// TIA Portal project "BangTai" (V17)

(* hardware
DEVICE "S7-1200 station_1"  S7-1200 Station
   slot 0: "Rack_0"  S7-1200 Rack  Rack  V1.0
   slot 1: "PLC _1"  CPU 1214C AC/DC/Rly  6ES7 214-1BG40-0XB0  V4.5
*)

// ===== PLC "PLC _1"  CPU 1214C AC/DC/Rly =====

VAR_GLOBAL   // PLC tag table "AO"
   "AQ_WeighConveyor.SpeedCMD" AT %QW0 : Int;
   "AQ_NormalConveyor.SpeedCMD" AT %QW2 : Int;
END_VAR

VAR_GLOBAL   // PLC tag table "AI"
   "AI_Weigh" AT %IW0 : Int;
   "AI_WeighConveyor.Speed" AT %IW2 : Int;
   "AI_NormalConveyor" AT %IW4 : Int;
END_VAR

VAR_GLOBAL   // PLC tag table "DO"
   "DO_WeighConveyor.CMD" AT %I7.0 : Bool;
   "DO_NormalConveyor.CMD" AT %I7.1 : Bool;
END_VAR

VAR_GLOBAL   // PLC tag table "DI"
   "DI_WeighConveyor.Run" AT %I6.0 : Bool;
   "DI_WeighConveyor.Fault" AT %I6.1 : Bool;
   "DI_WeighConveyor.Remote" AT %I6.2 : Bool;
   "DI_NormalConveyor.Run" AT %I6.3 : Bool;
   "DI_NormalConveyor.Fault" AT %I6.4 : Bool;
   "DI_NormalConveyor.Remote" AT %I6.5 : Bool;
   "DI_Oject" AT %I6.6 : Bool;
   "DI_WrongObject" AT %I6.7 : Bool;
END_VAR

TYPE "Sensor"
   STRUCT
      High_Value : Real;
      Low_Value : Real;
      Ratio : Real;
      Bias : Real;
      Real_Value : Real;
      HLM : Real;
      LLM : Real;
      HLM_Auxiliary : Real;
      LLM_Auxiliary : Real;
      Input_Error : Bool;
      Sensor_Error : Bool;
      Alarm_HLM : Bool;
      Alarm_LLM : Bool;
   END_STRUCT;
END_TYPE

TYPE "Motor_VDF"
   STRUCT
      Ctrl_Mode : Int;   // 0-Stop; 1-Manual; 2-Auto
      Enable : Bool;
      Lock : Bool;
      Manual_Lock : Bool;
      Status : Int;
      Runtime_60s : Int;
      Runtime_h : Int;
      Runtime_m : Int;
      Runtime_s : Int;
      P : Real;
      I : Real;
      D : Real;
      "Speed.RealValue" : Real;   // Gia tri doc tu bien tan
      "Speed.WriteHLM(Hz)" : Real;   // Gia tri tan so out Low
      "Speed.WriteLLM(Hz)" : Real;   // Gia tri tan so out High
      "Speed.Manual(Hz)" : Real;   // Gia tri tan so chay tay
      "Speed.WriteHLM(%)" : Real;   // Gia tri dung cho khoi PID 0->100 %
      "Speed.WriteLLM(%)" : Real;   // Gia tri tan so out High
      "Speed.Manual(%)" : Real;   // Gia tri tan so chay tay
      "ReadSpeed.Ratio" : Real;
      "ReadSpeed.Bias" : Real;
   END_STRUCT;
END_TYPE

TYPE "Motor_Normal"
   STRUCT
      Ctrl_Mode : Int;   // 0-Stop; 1-Manual; 2-Auto
      Enable : Bool;
      Lock : Bool;
      Manual_Lock : Bool;
      Status : Int;   // -1: Fault, 0:Stop, 1:Run
      Runtime_60s : Int;
      Runtime_h : Int;
      Runtime_m : Int;
      Runtime_s : Int;
   END_STRUCT;
END_TYPE

// folder: DataBlock

DATA_BLOCK "DB_READ_ABALOG"   // DB1
{ S7_Optimized_Access := 'TRUE' }
VERSION : 0.1
   VAR
      Weigh : "Sensor";
      sensor_weigh : Bool;
      sensor_wrong_object : Bool;
   END_VAR
BEGIN
END_DATA_BLOCK

DATA_BLOCK "DB_Conveyor"   // DB2
{ S7_Optimized_Access := 'TRUE' }
VERSION : 0.1
   VAR
      weigh_conveyor : "Motor_VDF";
      normal_conveyor : "Motor_VDF";
   END_VAR
BEGIN
END_DATA_BLOCK

// folder: (top level)

FUNCTION "FC_READ_ANALOG" : Void   // FC2, LAD
{ S7_Optimized_Access := 'TRUE' }
VERSION : 0.1
BEGIN

REGION Network 1: Đọc giá trị tốc độ băng tải cân
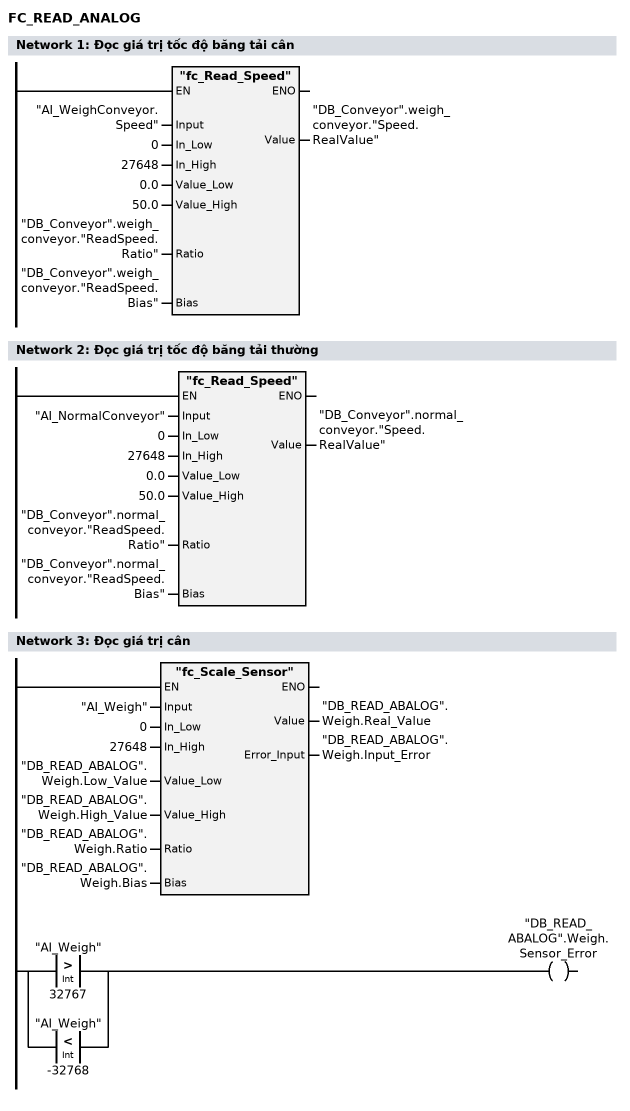
   RUNG wire#powerrail
      "fc_Read_Speed"(Input := "AI_WeighConveyor.Speed", In_Low := 0, In_High := 27648, Value_Low := 0.0, Value_High := 50.0, Ratio := "DB_Conveyor".weigh_conveyor."ReadSpeed.Ratio", Bias := "DB_Conveyor".weigh_conveyor."ReadSpeed.Bias", Value => "DB_Conveyor".weigh_conveyor."Speed.RealValue")
   END_RUNG
   // the same network as SCL:
   "fc_Read_Speed"(Input := "AI_WeighConveyor.Speed",
                   In_Low := 0,
                   In_High := 27648,
                   Value_Low := 0.0,
                   Value_High := 50.0,
                   Ratio := "DB_Conveyor".weigh_conveyor."ReadSpeed.Ratio",
                   Bias := "DB_Conveyor".weigh_conveyor."ReadSpeed.Bias",
                   Value => "DB_Conveyor".weigh_conveyor."Speed.RealValue");
END_REGION

REGION Network 2: Đọc giá trị tốc độ băng tải thường
   RUNG wire#powerrail
      "fc_Read_Speed"(Input := "AI_NormalConveyor", In_Low := 0, In_High := 27648, Value_Low := 0.0, Value_High := 50.0, Ratio := "DB_Conveyor".normal_conveyor."ReadSpeed.Ratio", Bias := "DB_Conveyor".normal_conveyor."ReadSpeed.Bias", Value => "DB_Conveyor".normal_conveyor."Speed.RealValue")
   END_RUNG
   // the same network as SCL:
   "fc_Read_Speed"(Input := "AI_NormalConveyor",
                   In_Low := 0,
                   In_High := 27648,
                   Value_Low := 0.0,
                   Value_High := 50.0,
                   Ratio := "DB_Conveyor".normal_conveyor."ReadSpeed.Ratio",
                   Bias := "DB_Conveyor".normal_conveyor."ReadSpeed.Bias",
                   Value => "DB_Conveyor".normal_conveyor."Speed.RealValue");
END_REGION

REGION Network 3: Đọc giá trị cân
   RUNG wire#powerrail
      "fc_Scale_Sensor"(Input := "AI_Weigh", In_Low := 0, In_High := 27648, Value_Low := "DB_READ_ABALOG".Weigh.Low_Value, Value_High := "DB_READ_ABALOG".Weigh.High_Value, Ratio := "DB_READ_ABALOG".Weigh.Ratio, Bias := "DB_READ_ABALOG".Weigh.Bias, Value => "DB_READ_ABALOG".Weigh.Real_Value, Error_Input => "DB_READ_ABALOG".Weigh.Input_Error)
   END_RUNG
   RUNG wire#powerrail
      { S7_Templates := "SrcType := Int" } GT_Contact(in1 := "AI_Weigh", in2 := 32767)
      wire#w1
      Coil( "DB_READ_ABALOG".Weigh.Sensor_Error )
   END_RUNG
   RUNG wire#powerrail
      { S7_Templates := "SrcType := Int" } LT_Contact(in1 := "AI_Weigh", in2 := -32768)
   END_RUNG wire#w1
   // the same network as SCL:
   "fc_Scale_Sensor"(Input := "AI_Weigh",
                     In_Low := 0,
                     In_High := 27648,
                     Value_Low := "DB_READ_ABALOG".Weigh.Low_Value,
                     Value_High := "DB_READ_ABALOG".Weigh.High_Value,
                     Ratio := "DB_READ_ABALOG".Weigh.Ratio,
                     Bias := "DB_READ_ABALOG".Weigh.Bias,
                     Value => "DB_READ_ABALOG".Weigh.Real_Value,
                     Error_Input => "DB_READ_ABALOG".Weigh.Input_Error);
   "DB_READ_ABALOG".Weigh.Sensor_Error := ("AI_Weigh" > 32767) OR ("AI_Weigh" < (-32768));
END_REGION
END_FUNCTION

FUNCTION "FC_ALARM" : Void   // FC3, LAD
{ S7_Optimized_Access := 'TRUE' }
VERSION : 0.1
BEGIN

REGION Network 1: Canh bao ap suat buong dot cao
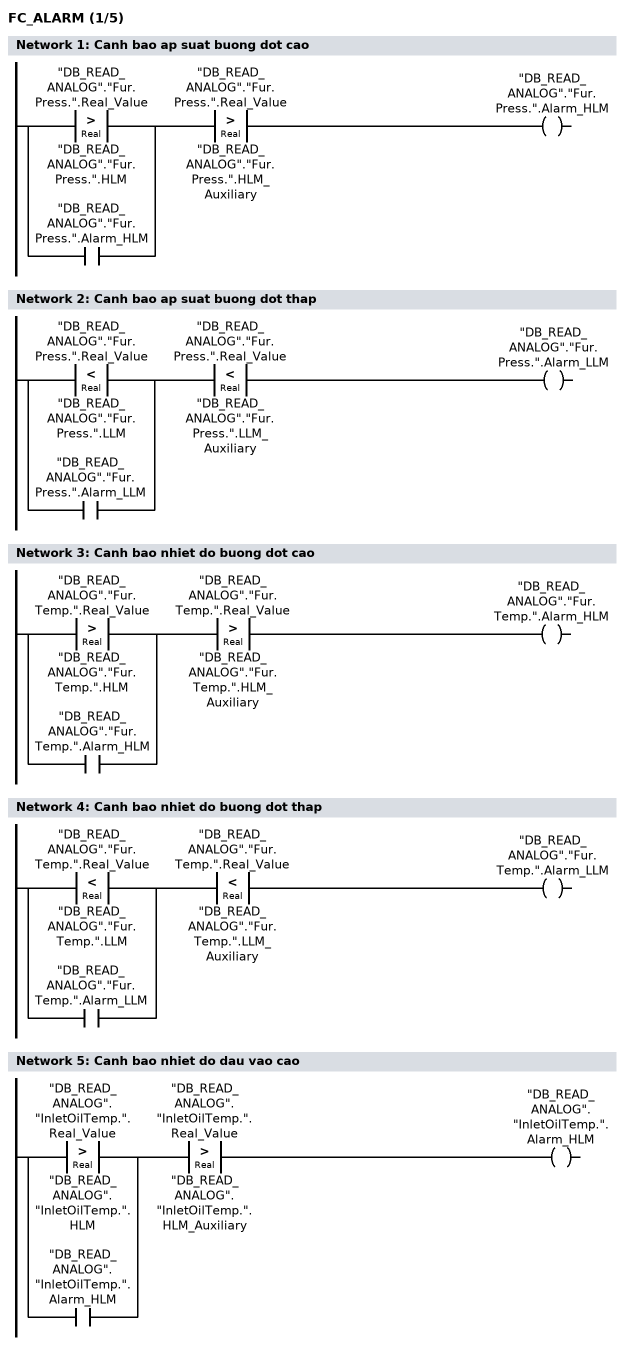
   RUNG wire#powerrail
      { S7_Templates := "SrcType := Real" } GT_Contact(in1 := "DB_READ_ANALOG"."Fur.Press.".Real_Value, in2 := "DB_READ_ANALOG"."Fur.Press.".HLM)
      wire#w1
      { S7_Templates := "SrcType := Real" } GT_Contact(in1 := "DB_READ_ANALOG"."Fur.Press.".Real_Value, in2 := "DB_READ_ANALOG"."Fur.Press.".HLM_Auxiliary)
      Coil( "DB_READ_ANALOG"."Fur.Press.".Alarm_HLM )
   END_RUNG
   RUNG wire#powerrail
      Contact( "DB_READ_ANALOG"."Fur.Press.".Alarm_HLM )
   END_RUNG wire#w1
   // the same network as SCL:
   "DB_READ_ANALOG"."Fur.Press.".Alarm_HLM := (("DB_READ_ANALOG"."Fur.Press.".Real_Value > "DB_READ_ANALOG"."Fur.Press.".HLM) OR "DB_READ_ANALOG"."Fur.Press.".Alarm_HLM) AND ("DB_READ_ANALOG"."Fur.Press.".Real_Value > "DB_READ_ANALOG"."Fur.Press.".HLM_Auxiliary);
END_REGION

REGION Network 2: Canh bao ap suat buong dot thap
   RUNG wire#powerrail
      { S7_Templates := "SrcType := Real" } LT_Contact(in1 := "DB_READ_ANALOG"."Fur.Press.".Real_Value, in2 := "DB_READ_ANALOG"."Fur.Press.".LLM)
      wire#w1
      { S7_Templates := "SrcType := Real" } LT_Contact(in1 := "DB_READ_ANALOG"."Fur.Press.".Real_Value, in2 := "DB_READ_ANALOG"."Fur.Press.".LLM_Auxiliary)
      Coil( "DB_READ_ANALOG"."Fur.Press.".Alarm_LLM )
   END_RUNG
   RUNG wire#powerrail
      Contact( "DB_READ_ANALOG"."Fur.Press.".Alarm_LLM )
   END_RUNG wire#w1
   // the same network as SCL:
   "DB_READ_ANALOG"."Fur.Press.".Alarm_LLM := (("DB_READ_ANALOG"."Fur.Press.".Real_Value < "DB_READ_ANALOG"."Fur.Press.".LLM) OR "DB_READ_ANALOG"."Fur.Press.".Alarm_LLM) AND ("DB_READ_ANALOG"."Fur.Press.".Real_Value < "DB_READ_ANALOG"."Fur.Press.".LLM_Auxiliary);
END_REGION

REGION Network 3: Canh bao nhiet do buong dot cao
   RUNG wire#powerrail
      { S7_Templates := "SrcType := Real" } GT_Contact(in1 := "DB_READ_ANALOG"."Fur.Temp.".Real_Value, in2 := "DB_READ_ANALOG"."Fur.Temp.".HLM)
      wire#w1
      { S7_Templates := "SrcType := Real" } GT_Contact(in1 := "DB_READ_ANALOG"."Fur.Temp.".Real_Value, in2 := "DB_READ_ANALOG"."Fur.Temp.".HLM_Auxiliary)
      Coil( "DB_READ_ANALOG"."Fur.Temp.".Alarm_HLM )
   END_RUNG
   RUNG wire#powerrail
      Contact( "DB_READ_ANALOG"."Fur.Temp.".Alarm_HLM )
   END_RUNG wire#w1
   // the same network as SCL:
   "DB_READ_ANALOG"."Fur.Temp.".Alarm_HLM := (("DB_READ_ANALOG"."Fur.Temp.".Real_Value > "DB_READ_ANALOG"."Fur.Temp.".HLM) OR "DB_READ_ANALOG"."Fur.Temp.".Alarm_HLM) AND ("DB_READ_ANALOG"."Fur.Temp.".Real_Value > "DB_READ_ANALOG"."Fur.Temp.".HLM_Auxiliary);
END_REGION

REGION Network 4: Canh bao nhiet do buong dot thap
   RUNG wire#powerrail
      { S7_Templates := "SrcType := Real" } LT_Contact(in1 := "DB_READ_ANALOG"."Fur.Temp.".Real_Value, in2 := "DB_READ_ANALOG"."Fur.Temp.".LLM)
      wire#w1
      { S7_Templates := "SrcType := Real" } LT_Contact(in1 := "DB_READ_ANALOG"."Fur.Temp.".Real_Value, in2 := "DB_READ_ANALOG"."Fur.Temp.".LLM_Auxiliary)
      Coil( "DB_READ_ANALOG"."Fur.Temp.".Alarm_LLM )
   END_RUNG
   RUNG wire#powerrail
      Contact( "DB_READ_ANALOG"."Fur.Temp.".Alarm_LLM )
   END_RUNG wire#w1
   // the same network as SCL:
   "DB_READ_ANALOG"."Fur.Temp.".Alarm_LLM := (("DB_READ_ANALOG"."Fur.Temp.".Real_Value < "DB_READ_ANALOG"."Fur.Temp.".LLM) OR "DB_READ_ANALOG"."Fur.Temp.".Alarm_LLM) AND ("DB_READ_ANALOG"."Fur.Temp.".Real_Value < "DB_READ_ANALOG"."Fur.Temp.".LLM_Auxiliary);
END_REGION

REGION Network 5: Canh bao nhiet do dau vao cao
   RUNG wire#powerrail
      { S7_Templates := "SrcType := Real" } GT_Contact(in1 := "DB_READ_ANALOG"."InletOilTemp.".Real_Value, in2 := "DB_READ_ANALOG"."InletOilTemp.".HLM)
      wire#w1
      { S7_Templates := "SrcType := Real" } GT_Contact(in1 := "DB_READ_ANALOG"."InletOilTemp.".Real_Value, in2 := "DB_READ_ANALOG"."InletOilTemp.".HLM_Auxiliary)
      Coil( "DB_READ_ANALOG"."InletOilTemp.".Alarm_HLM )
   END_RUNG
   RUNG wire#powerrail
      Contact( "DB_READ_ANALOG"."InletOilTemp.".Alarm_HLM )
   END_RUNG wire#w1
   // the same network as SCL:
   "DB_READ_ANALOG"."InletOilTemp.".Alarm_HLM := (("DB_READ_ANALOG"."InletOilTemp.".Real_Value > "DB_READ_ANALOG"."InletOilTemp.".HLM) OR "DB_READ_ANALOG"."InletOilTemp.".Alarm_HLM) AND ("DB_READ_ANALOG"."InletOilTemp.".Real_Value > "DB_READ_ANALOG"."InletOilTemp.".HLM_Auxiliary);
END_REGION

REGION Network 6: Canh bao nhiet do dau vao thap
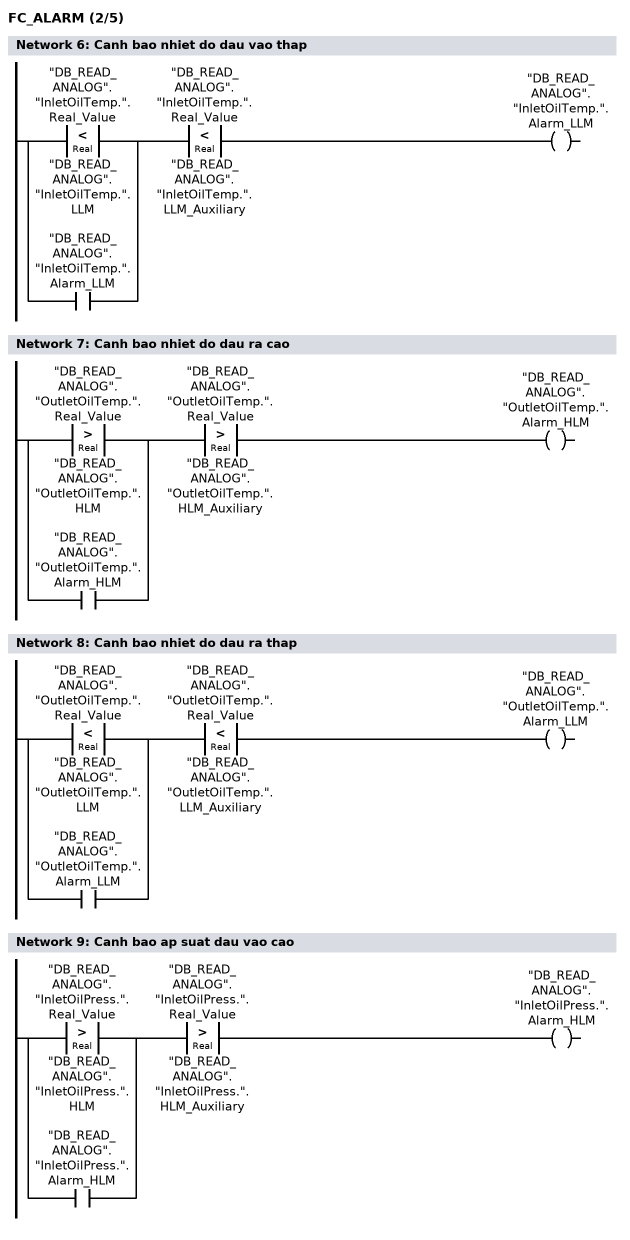
   RUNG wire#powerrail
      { S7_Templates := "SrcType := Real" } LT_Contact(in1 := "DB_READ_ANALOG"."InletOilTemp.".Real_Value, in2 := "DB_READ_ANALOG"."InletOilTemp.".LLM)
      wire#w1
      { S7_Templates := "SrcType := Real" } LT_Contact(in1 := "DB_READ_ANALOG"."InletOilTemp.".Real_Value, in2 := "DB_READ_ANALOG"."InletOilTemp.".LLM_Auxiliary)
      Coil( "DB_READ_ANALOG"."InletOilTemp.".Alarm_LLM )
   END_RUNG
   RUNG wire#powerrail
      Contact( "DB_READ_ANALOG"."InletOilTemp.".Alarm_LLM )
   END_RUNG wire#w1
   // the same network as SCL:
   "DB_READ_ANALOG"."InletOilTemp.".Alarm_LLM := (("DB_READ_ANALOG"."InletOilTemp.".Real_Value < "DB_READ_ANALOG"."InletOilTemp.".LLM) OR "DB_READ_ANALOG"."InletOilTemp.".Alarm_LLM) AND ("DB_READ_ANALOG"."InletOilTemp.".Real_Value < "DB_READ_ANALOG"."InletOilTemp.".LLM_Auxiliary);
END_REGION

REGION Network 7: Canh bao nhiet do dau ra cao
   RUNG wire#powerrail
      { S7_Templates := "SrcType := Real" } GT_Contact(in1 := "DB_READ_ANALOG"."OutletOilTemp.".Real_Value, in2 := "DB_READ_ANALOG"."OutletOilTemp.".HLM)
      wire#w1
      { S7_Templates := "SrcType := Real" } GT_Contact(in1 := "DB_READ_ANALOG"."OutletOilTemp.".Real_Value, in2 := "DB_READ_ANALOG"."OutletOilTemp.".HLM_Auxiliary)
      Coil( "DB_READ_ANALOG"."OutletOilTemp.".Alarm_HLM )
   END_RUNG
   RUNG wire#powerrail
      Contact( "DB_READ_ANALOG"."OutletOilTemp.".Alarm_HLM )
   END_RUNG wire#w1
   // the same network as SCL:
   "DB_READ_ANALOG"."OutletOilTemp.".Alarm_HLM := (("DB_READ_ANALOG"."OutletOilTemp.".Real_Value > "DB_READ_ANALOG"."OutletOilTemp.".HLM) OR "DB_READ_ANALOG"."OutletOilTemp.".Alarm_HLM) AND ("DB_READ_ANALOG"."OutletOilTemp.".Real_Value > "DB_READ_ANALOG"."OutletOilTemp.".HLM_Auxiliary);
END_REGION

REGION Network 8: Canh bao nhiet do dau ra thap
   RUNG wire#powerrail
      { S7_Templates := "SrcType := Real" } LT_Contact(in1 := "DB_READ_ANALOG"."OutletOilTemp.".Real_Value, in2 := "DB_READ_ANALOG"."OutletOilTemp.".LLM)
      wire#w1
      { S7_Templates := "SrcType := Real" } LT_Contact(in1 := "DB_READ_ANALOG"."OutletOilTemp.".Real_Value, in2 := "DB_READ_ANALOG"."OutletOilTemp.".LLM_Auxiliary)
      Coil( "DB_READ_ANALOG"."OutletOilTemp.".Alarm_LLM )
   END_RUNG
   RUNG wire#powerrail
      Contact( "DB_READ_ANALOG"."OutletOilTemp.".Alarm_LLM )
   END_RUNG wire#w1
   // the same network as SCL:
   "DB_READ_ANALOG"."OutletOilTemp.".Alarm_LLM := (("DB_READ_ANALOG"."OutletOilTemp.".Real_Value < "DB_READ_ANALOG"."OutletOilTemp.".LLM) OR "DB_READ_ANALOG"."OutletOilTemp.".Alarm_LLM) AND ("DB_READ_ANALOG"."OutletOilTemp.".Real_Value < "DB_READ_ANALOG"."OutletOilTemp.".LLM_Auxiliary);
END_REGION

REGION Network 9: Canh bao ap suat dau vao cao
   RUNG wire#powerrail
      { S7_Templates := "SrcType := Real" } GT_Contact(in1 := "DB_READ_ANALOG"."InletOilPress.".Real_Value, in2 := "DB_READ_ANALOG"."InletOilPress.".HLM)
      wire#w1
      { S7_Templates := "SrcType := Real" } GT_Contact(in1 := "DB_READ_ANALOG"."InletOilPress.".Real_Value, in2 := "DB_READ_ANALOG"."InletOilPress.".HLM_Auxiliary)
      Coil( "DB_READ_ANALOG"."InletOilPress.".Alarm_HLM )
   END_RUNG
   RUNG wire#powerrail
      Contact( "DB_READ_ANALOG"."InletOilPress.".Alarm_HLM )
   END_RUNG wire#w1
   // the same network as SCL:
   "DB_READ_ANALOG"."InletOilPress.".Alarm_HLM := (("DB_READ_ANALOG"."InletOilPress.".Real_Value > "DB_READ_ANALOG"."InletOilPress.".HLM) OR "DB_READ_ANALOG"."InletOilPress.".Alarm_HLM) AND ("DB_READ_ANALOG"."InletOilPress.".Real_Value > "DB_READ_ANALOG"."InletOilPress.".HLM_Auxiliary);
END_REGION

REGION Network 10: Canh bao ap suat dau vao thap
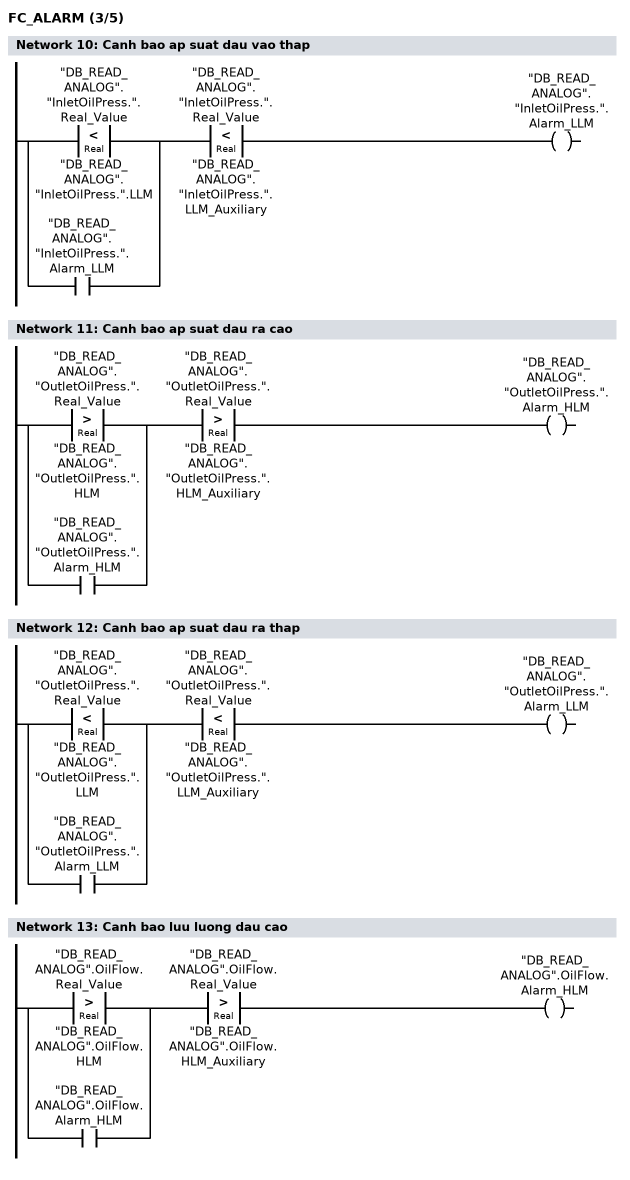
   RUNG wire#powerrail
      { S7_Templates := "SrcType := Real" } LT_Contact(in1 := "DB_READ_ANALOG"."InletOilPress.".Real_Value, in2 := "DB_READ_ANALOG"."InletOilPress.".LLM)
      wire#w1
      { S7_Templates := "SrcType := Real" } LT_Contact(in1 := "DB_READ_ANALOG"."InletOilPress.".Real_Value, in2 := "DB_READ_ANALOG"."InletOilPress.".LLM_Auxiliary)
      Coil( "DB_READ_ANALOG"."InletOilPress.".Alarm_LLM )
   END_RUNG
   RUNG wire#powerrail
      Contact( "DB_READ_ANALOG"."InletOilPress.".Alarm_LLM )
   END_RUNG wire#w1
   // the same network as SCL:
   "DB_READ_ANALOG"."InletOilPress.".Alarm_LLM := (("DB_READ_ANALOG"."InletOilPress.".Real_Value < "DB_READ_ANALOG"."InletOilPress.".LLM) OR "DB_READ_ANALOG"."InletOilPress.".Alarm_LLM) AND ("DB_READ_ANALOG"."InletOilPress.".Real_Value < "DB_READ_ANALOG"."InletOilPress.".LLM_Auxiliary);
END_REGION

REGION Network 11: Canh bao ap suat dau ra cao
   RUNG wire#powerrail
      { S7_Templates := "SrcType := Real" } GT_Contact(in1 := "DB_READ_ANALOG"."OutletOilPress.".Real_Value, in2 := "DB_READ_ANALOG"."OutletOilPress.".HLM)
      wire#w1
      { S7_Templates := "SrcType := Real" } GT_Contact(in1 := "DB_READ_ANALOG"."OutletOilPress.".Real_Value, in2 := "DB_READ_ANALOG"."OutletOilPress.".HLM_Auxiliary)
      Coil( "DB_READ_ANALOG"."OutletOilPress.".Alarm_HLM )
   END_RUNG
   RUNG wire#powerrail
      Contact( "DB_READ_ANALOG"."OutletOilPress.".Alarm_HLM )
   END_RUNG wire#w1
   // the same network as SCL:
   "DB_READ_ANALOG"."OutletOilPress.".Alarm_HLM := (("DB_READ_ANALOG"."OutletOilPress.".Real_Value > "DB_READ_ANALOG"."OutletOilPress.".HLM) OR "DB_READ_ANALOG"."OutletOilPress.".Alarm_HLM) AND ("DB_READ_ANALOG"."OutletOilPress.".Real_Value > "DB_READ_ANALOG"."OutletOilPress.".HLM_Auxiliary);
END_REGION

REGION Network 12: Canh bao ap suat dau ra thap
   RUNG wire#powerrail
      { S7_Templates := "SrcType := Real" } LT_Contact(in1 := "DB_READ_ANALOG"."OutletOilPress.".Real_Value, in2 := "DB_READ_ANALOG"."OutletOilPress.".LLM)
      wire#w1
      { S7_Templates := "SrcType := Real" } LT_Contact(in1 := "DB_READ_ANALOG"."OutletOilPress.".Real_Value, in2 := "DB_READ_ANALOG"."OutletOilPress.".LLM_Auxiliary)
      Coil( "DB_READ_ANALOG"."OutletOilPress.".Alarm_LLM )
   END_RUNG
   RUNG wire#powerrail
      Contact( "DB_READ_ANALOG"."OutletOilPress.".Alarm_LLM )
   END_RUNG wire#w1
   // the same network as SCL:
   "DB_READ_ANALOG"."OutletOilPress.".Alarm_LLM := (("DB_READ_ANALOG"."OutletOilPress.".Real_Value < "DB_READ_ANALOG"."OutletOilPress.".LLM) OR "DB_READ_ANALOG"."OutletOilPress.".Alarm_LLM) AND ("DB_READ_ANALOG"."OutletOilPress.".Real_Value < "DB_READ_ANALOG"."OutletOilPress.".LLM_Auxiliary);
END_REGION

REGION Network 13: Canh bao luu luong dau cao
   RUNG wire#powerrail
      { S7_Templates := "SrcType := Real" } GT_Contact(in1 := "DB_READ_ANALOG".OilFlow.Real_Value, in2 := "DB_READ_ANALOG".OilFlow.HLM)
      wire#w1
      { S7_Templates := "SrcType := Real" } GT_Contact(in1 := "DB_READ_ANALOG".OilFlow.Real_Value, in2 := "DB_READ_ANALOG".OilFlow.HLM_Auxiliary)
      Coil( "DB_READ_ANALOG".OilFlow.Alarm_HLM )
   END_RUNG
   RUNG wire#powerrail
      Contact( "DB_READ_ANALOG".OilFlow.Alarm_HLM )
   END_RUNG wire#w1
   // the same network as SCL:
   "DB_READ_ANALOG".OilFlow.Alarm_HLM := (("DB_READ_ANALOG".OilFlow.Real_Value > "DB_READ_ANALOG".OilFlow.HLM) OR "DB_READ_ANALOG".OilFlow.Alarm_HLM) AND ("DB_READ_ANALOG".OilFlow.Real_Value > "DB_READ_ANALOG".OilFlow.HLM_Auxiliary);
END_REGION

REGION Network 14: Canh bao luu luong dau thap
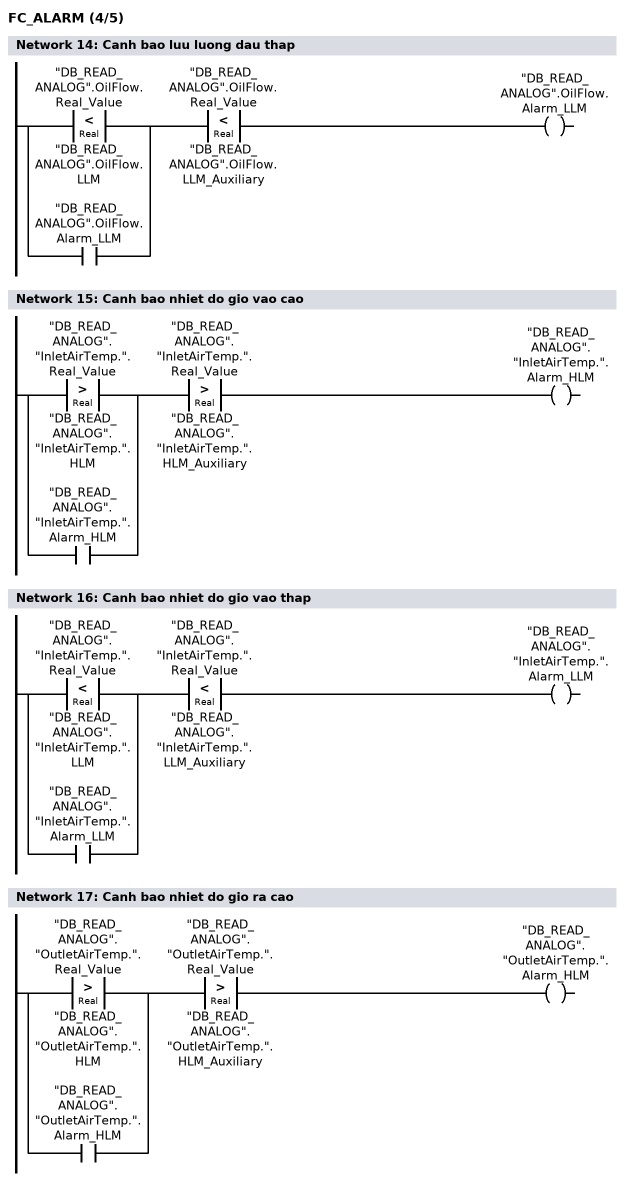
   RUNG wire#powerrail
      { S7_Templates := "SrcType := Real" } LT_Contact(in1 := "DB_READ_ANALOG".OilFlow.Real_Value, in2 := "DB_READ_ANALOG".OilFlow.LLM)
      wire#w1
      { S7_Templates := "SrcType := Real" } LT_Contact(in1 := "DB_READ_ANALOG".OilFlow.Real_Value, in2 := "DB_READ_ANALOG".OilFlow.LLM_Auxiliary)
      Coil( "DB_READ_ANALOG".OilFlow.Alarm_LLM )
   END_RUNG
   RUNG wire#powerrail
      Contact( "DB_READ_ANALOG".OilFlow.Alarm_LLM )
   END_RUNG wire#w1
   // the same network as SCL:
   "DB_READ_ANALOG".OilFlow.Alarm_LLM := (("DB_READ_ANALOG".OilFlow.Real_Value < "DB_READ_ANALOG".OilFlow.LLM) OR "DB_READ_ANALOG".OilFlow.Alarm_LLM) AND ("DB_READ_ANALOG".OilFlow.Real_Value < "DB_READ_ANALOG".OilFlow.LLM_Auxiliary);
END_REGION

REGION Network 15: Canh bao nhiet do gio vao cao
   RUNG wire#powerrail
      { S7_Templates := "SrcType := Real" } GT_Contact(in1 := "DB_READ_ANALOG"."InletAirTemp.".Real_Value, in2 := "DB_READ_ANALOG"."InletAirTemp.".HLM)
      wire#w1
      { S7_Templates := "SrcType := Real" } GT_Contact(in1 := "DB_READ_ANALOG"."InletAirTemp.".Real_Value, in2 := "DB_READ_ANALOG"."InletAirTemp.".HLM_Auxiliary)
      Coil( "DB_READ_ANALOG"."InletAirTemp.".Alarm_HLM )
   END_RUNG
   RUNG wire#powerrail
      Contact( "DB_READ_ANALOG"."InletAirTemp.".Alarm_HLM )
   END_RUNG wire#w1
   // the same network as SCL:
   "DB_READ_ANALOG"."InletAirTemp.".Alarm_HLM := (("DB_READ_ANALOG"."InletAirTemp.".Real_Value > "DB_READ_ANALOG"."InletAirTemp.".HLM) OR "DB_READ_ANALOG"."InletAirTemp.".Alarm_HLM) AND ("DB_READ_ANALOG"."InletAirTemp.".Real_Value > "DB_READ_ANALOG"."InletAirTemp.".HLM_Auxiliary);
END_REGION

REGION Network 16: Canh bao nhiet do gio vao thap
   RUNG wire#powerrail
      { S7_Templates := "SrcType := Real" } LT_Contact(in1 := "DB_READ_ANALOG"."InletAirTemp.".Real_Value, in2 := "DB_READ_ANALOG"."InletAirTemp.".LLM)
      wire#w1
      { S7_Templates := "SrcType := Real" } LT_Contact(in1 := "DB_READ_ANALOG"."InletAirTemp.".Real_Value, in2 := "DB_READ_ANALOG"."InletAirTemp.".LLM_Auxiliary)
      Coil( "DB_READ_ANALOG"."InletAirTemp.".Alarm_LLM )
   END_RUNG
   RUNG wire#powerrail
      Contact( "DB_READ_ANALOG"."InletAirTemp.".Alarm_LLM )
   END_RUNG wire#w1
   // the same network as SCL:
   "DB_READ_ANALOG"."InletAirTemp.".Alarm_LLM := (("DB_READ_ANALOG"."InletAirTemp.".Real_Value < "DB_READ_ANALOG"."InletAirTemp.".LLM) OR "DB_READ_ANALOG"."InletAirTemp.".Alarm_LLM) AND ("DB_READ_ANALOG"."InletAirTemp.".Real_Value < "DB_READ_ANALOG"."InletAirTemp.".LLM_Auxiliary);
END_REGION

REGION Network 17: Canh bao nhiet do gio ra cao
   RUNG wire#powerrail
      { S7_Templates := "SrcType := Real" } GT_Contact(in1 := "DB_READ_ANALOG"."OutletAirTemp.".Real_Value, in2 := "DB_READ_ANALOG"."OutletAirTemp.".HLM)
      wire#w1
      { S7_Templates := "SrcType := Real" } GT_Contact(in1 := "DB_READ_ANALOG"."OutletAirTemp.".Real_Value, in2 := "DB_READ_ANALOG"."OutletAirTemp.".HLM_Auxiliary)
      Coil( "DB_READ_ANALOG"."OutletAirTemp.".Alarm_HLM )
   END_RUNG
   RUNG wire#powerrail
      Contact( "DB_READ_ANALOG"."OutletAirTemp.".Alarm_HLM )
   END_RUNG wire#w1
   // the same network as SCL:
   "DB_READ_ANALOG"."OutletAirTemp.".Alarm_HLM := (("DB_READ_ANALOG"."OutletAirTemp.".Real_Value > "DB_READ_ANALOG"."OutletAirTemp.".HLM) OR "DB_READ_ANALOG"."OutletAirTemp.".Alarm_HLM) AND ("DB_READ_ANALOG"."OutletAirTemp.".Real_Value > "DB_READ_ANALOG"."OutletAirTemp.".HLM_Auxiliary);
END_REGION

REGION Network 18: Canh bao nhiet do gio ra thap
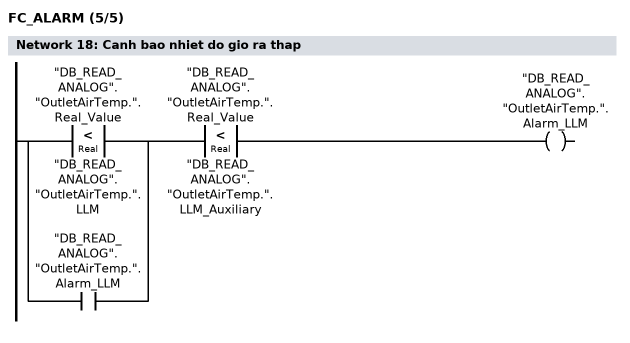
   RUNG wire#powerrail
      { S7_Templates := "SrcType := Real" } LT_Contact(in1 := "DB_READ_ANALOG"."OutletAirTemp.".Real_Value, in2 := "DB_READ_ANALOG"."OutletAirTemp.".LLM)
      wire#w1
      { S7_Templates := "SrcType := Real" } LT_Contact(in1 := "DB_READ_ANALOG"."OutletAirTemp.".Real_Value, in2 := "DB_READ_ANALOG"."OutletAirTemp.".LLM_Auxiliary)
      Coil( "DB_READ_ANALOG"."OutletAirTemp.".Alarm_LLM )
   END_RUNG
   RUNG wire#powerrail
      Contact( "DB_READ_ANALOG"."OutletAirTemp.".Alarm_LLM )
   END_RUNG wire#w1
   // the same network as SCL:
   "DB_READ_ANALOG"."OutletAirTemp.".Alarm_LLM := (("DB_READ_ANALOG"."OutletAirTemp.".Real_Value < "DB_READ_ANALOG"."OutletAirTemp.".LLM) OR "DB_READ_ANALOG"."OutletAirTemp.".Alarm_LLM) AND ("DB_READ_ANALOG"."OutletAirTemp.".Real_Value < "DB_READ_ANALOG"."OutletAirTemp.".LLM_Auxiliary);
END_REGION
END_FUNCTION

FUNCTION "FC_MOTOR" : Void   // FC4, LAD
{ S7_Optimized_Access := 'TRUE' }
VERSION : 0.1
BEGIN

REGION Network 1: IDF
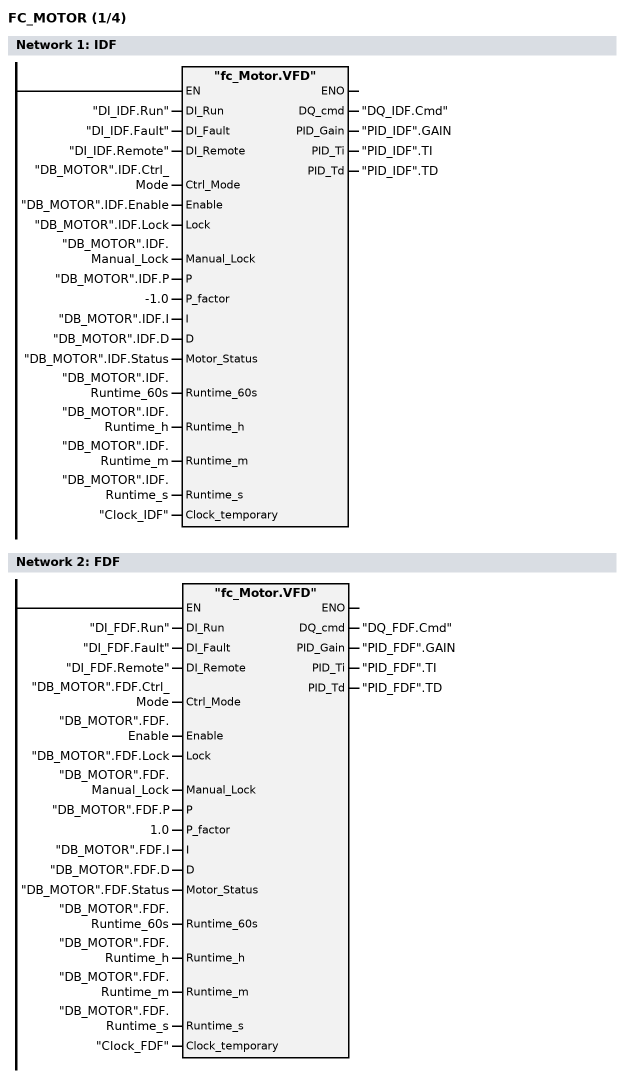
   RUNG wire#powerrail
      "fc_Motor.VFD"(DI_Run := "DI_IDF.Run", DI_Fault := "DI_IDF.Fault", DI_Remote := "DI_IDF.Remote", Ctrl_Mode := "DB_MOTOR".IDF.Ctrl_Mode, Enable := "DB_MOTOR".IDF.Enable, Lock := "DB_MOTOR".IDF.Lock, Manual_Lock := "DB_MOTOR".IDF.Manual_Lock, P := "DB_MOTOR".IDF.P, P_factor := -1.0, I := "DB_MOTOR".IDF.I, D := "DB_MOTOR".IDF.D, Motor_Status := "DB_MOTOR".IDF.Status, Runtime_60s := "DB_MOTOR".IDF.Runtime_60s, Runtime_h := "DB_MOTOR".IDF.Runtime_h, Runtime_m := "DB_MOTOR".IDF.Runtime_m, Runtime_s := "DB_MOTOR".IDF.Runtime_s, Clock_temporary := "Clock_IDF", DQ_cmd => "DQ_IDF.Cmd", PID_Gain => "PID_IDF".GAIN, PID_Ti => "PID_IDF".TI, PID_Td => "PID_IDF".TD)
   END_RUNG
   // the same network as SCL:
   "fc_Motor.VFD"(DI_Run := "DI_IDF.Run",
                  DI_Fault := "DI_IDF.Fault",
                  DI_Remote := "DI_IDF.Remote",
                  Ctrl_Mode := "DB_MOTOR".IDF.Ctrl_Mode,
                  Enable := "DB_MOTOR".IDF.Enable,
                  Lock := "DB_MOTOR".IDF.Lock,
                  Manual_Lock := "DB_MOTOR".IDF.Manual_Lock,
                  P := "DB_MOTOR".IDF.P,
                  P_factor := -1.0,
                  I := "DB_MOTOR".IDF.I,
                  D := "DB_MOTOR".IDF.D,
                  Motor_Status := "DB_MOTOR".IDF.Status,
                  Runtime_60s := "DB_MOTOR".IDF.Runtime_60s,
                  Runtime_h := "DB_MOTOR".IDF.Runtime_h,
                  Runtime_m := "DB_MOTOR".IDF.Runtime_m,
                  Runtime_s := "DB_MOTOR".IDF.Runtime_s,
                  Clock_temporary := "Clock_IDF",
                  DQ_cmd => "DQ_IDF.Cmd",
                  PID_Gain => "PID_IDF".GAIN,
                  PID_Ti => "PID_IDF".TI,
                  PID_Td => "PID_IDF".TD);
END_REGION

REGION Network 2: FDF
   RUNG wire#powerrail
      "fc_Motor.VFD"(DI_Run := "DI_FDF.Run", DI_Fault := "DI_FDF.Fault", DI_Remote := "DI_FDF.Remote", Ctrl_Mode := "DB_MOTOR".FDF.Ctrl_Mode, Enable := "DB_MOTOR".FDF.Enable, Lock := "DB_MOTOR".FDF.Lock, Manual_Lock := "DB_MOTOR".FDF.Manual_Lock, P := "DB_MOTOR".FDF.P, P_factor := 1.0, I := "DB_MOTOR".FDF.I, D := "DB_MOTOR".FDF.D, Motor_Status := "DB_MOTOR".FDF.Status, Runtime_60s := "DB_MOTOR".FDF.Runtime_60s, Runtime_h := "DB_MOTOR".FDF.Runtime_h, Runtime_m := "DB_MOTOR".FDF.Runtime_m, Runtime_s := "DB_MOTOR".FDF.Runtime_s, Clock_temporary := "Clock_FDF", DQ_cmd => "DQ_FDF.Cmd", PID_Gain => "PID_FDF".GAIN, PID_Ti => "PID_FDF".TI, PID_Td => "PID_FDF".TD)
   END_RUNG
   // the same network as SCL:
   "fc_Motor.VFD"(DI_Run := "DI_FDF.Run",
                  DI_Fault := "DI_FDF.Fault",
                  DI_Remote := "DI_FDF.Remote",
                  Ctrl_Mode := "DB_MOTOR".FDF.Ctrl_Mode,
                  Enable := "DB_MOTOR".FDF.Enable,
                  Lock := "DB_MOTOR".FDF.Lock,
                  Manual_Lock := "DB_MOTOR".FDF.Manual_Lock,
                  P := "DB_MOTOR".FDF.P,
                  P_factor := 1.0,
                  I := "DB_MOTOR".FDF.I,
                  D := "DB_MOTOR".FDF.D,
                  Motor_Status := "DB_MOTOR".FDF.Status,
                  Runtime_60s := "DB_MOTOR".FDF.Runtime_60s,
                  Runtime_h := "DB_MOTOR".FDF.Runtime_h,
                  Runtime_m := "DB_MOTOR".FDF.Runtime_m,
                  Runtime_s := "DB_MOTOR".FDF.Runtime_s,
                  Clock_temporary := "Clock_FDF",
                  DQ_cmd => "DQ_FDF.Cmd",
                  PID_Gain => "PID_FDF".GAIN,
                  PID_Ti => "PID_FDF".TI,
                  PID_Td => "PID_FDF".TD);
END_REGION

REGION Network 3: CHG
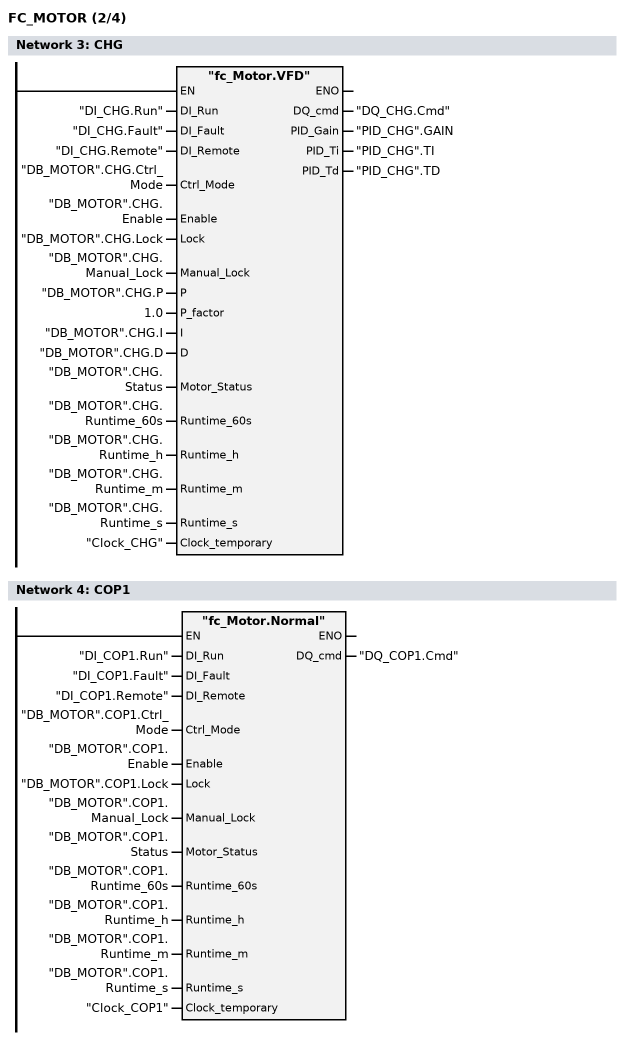
   RUNG wire#powerrail
      "fc_Motor.VFD"(DI_Run := "DI_CHG.Run", DI_Fault := "DI_CHG.Fault", DI_Remote := "DI_CHG.Remote", Ctrl_Mode := "DB_MOTOR".CHG.Ctrl_Mode, Enable := "DB_MOTOR".CHG.Enable, Lock := "DB_MOTOR".CHG.Lock, Manual_Lock := "DB_MOTOR".CHG.Manual_Lock, P := "DB_MOTOR".CHG.P, P_factor := 1.0, I := "DB_MOTOR".CHG.I, D := "DB_MOTOR".CHG.D, Motor_Status := "DB_MOTOR".CHG.Status, Runtime_60s := "DB_MOTOR".CHG.Runtime_60s, Runtime_h := "DB_MOTOR".CHG.Runtime_h, Runtime_m := "DB_MOTOR".CHG.Runtime_m, Runtime_s := "DB_MOTOR".CHG.Runtime_s, Clock_temporary := "Clock_CHG", DQ_cmd => "DQ_CHG.Cmd", PID_Gain => "PID_CHG".GAIN, PID_Ti => "PID_CHG".TI, PID_Td => "PID_CHG".TD)
   END_RUNG
   // the same network as SCL:
   "fc_Motor.VFD"(DI_Run := "DI_CHG.Run",
                  DI_Fault := "DI_CHG.Fault",
                  DI_Remote := "DI_CHG.Remote",
                  Ctrl_Mode := "DB_MOTOR".CHG.Ctrl_Mode,
                  Enable := "DB_MOTOR".CHG.Enable,
                  Lock := "DB_MOTOR".CHG.Lock,
                  Manual_Lock := "DB_MOTOR".CHG.Manual_Lock,
                  P := "DB_MOTOR".CHG.P,
                  P_factor := 1.0,
                  I := "DB_MOTOR".CHG.I,
                  D := "DB_MOTOR".CHG.D,
                  Motor_Status := "DB_MOTOR".CHG.Status,
                  Runtime_60s := "DB_MOTOR".CHG.Runtime_60s,
                  Runtime_h := "DB_MOTOR".CHG.Runtime_h,
                  Runtime_m := "DB_MOTOR".CHG.Runtime_m,
                  Runtime_s := "DB_MOTOR".CHG.Runtime_s,
                  Clock_temporary := "Clock_CHG",
                  DQ_cmd => "DQ_CHG.Cmd",
                  PID_Gain => "PID_CHG".GAIN,
                  PID_Ti => "PID_CHG".TI,
                  PID_Td => "PID_CHG".TD);
END_REGION

REGION Network 4: COP1
   RUNG wire#powerrail
      "fc_Motor.Normal"(DI_Run := "DI_COP1.Run", DI_Fault := "DI_COP1.Fault", DI_Remote := "DI_COP1.Remote", Ctrl_Mode := "DB_MOTOR".COP1.Ctrl_Mode, Enable := "DB_MOTOR".COP1.Enable, Lock := "DB_MOTOR".COP1.Lock, Manual_Lock := "DB_MOTOR".COP1.Manual_Lock, Motor_Status := "DB_MOTOR".COP1.Status, Runtime_60s := "DB_MOTOR".COP1.Runtime_60s, Runtime_h := "DB_MOTOR".COP1.Runtime_h, Runtime_m := "DB_MOTOR".COP1.Runtime_m, Runtime_s := "DB_MOTOR".COP1.Runtime_s, Clock_temporary := "Clock_COP1", DQ_cmd => "DQ_COP1.Cmd")
   END_RUNG
   // the same network as SCL:
   "fc_Motor.Normal"(DI_Run := "DI_COP1.Run",
                     DI_Fault := "DI_COP1.Fault",
                     DI_Remote := "DI_COP1.Remote",
                     Ctrl_Mode := "DB_MOTOR".COP1.Ctrl_Mode,
                     Enable := "DB_MOTOR".COP1.Enable,
                     Lock := "DB_MOTOR".COP1.Lock,
                     Manual_Lock := "DB_MOTOR".COP1.Manual_Lock,
                     Motor_Status := "DB_MOTOR".COP1.Status,
                     Runtime_60s := "DB_MOTOR".COP1.Runtime_60s,
                     Runtime_h := "DB_MOTOR".COP1.Runtime_h,
                     Runtime_m := "DB_MOTOR".COP1.Runtime_m,
                     Runtime_s := "DB_MOTOR".COP1.Runtime_s,
                     Clock_temporary := "Clock_COP1",
                     DQ_cmd => "DQ_COP1.Cmd");
END_REGION

REGION Network 5: COP2
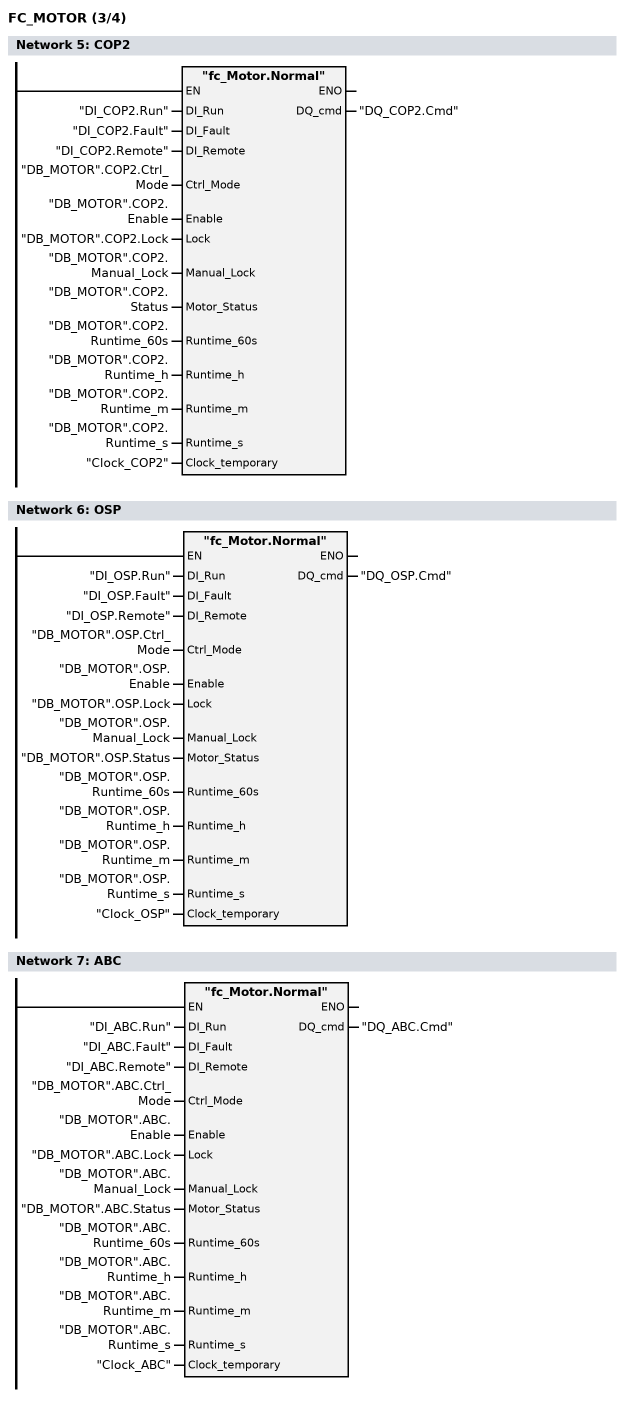
   RUNG wire#powerrail
      "fc_Motor.Normal"(DI_Run := "DI_COP2.Run", DI_Fault := "DI_COP2.Fault", DI_Remote := "DI_COP2.Remote", Ctrl_Mode := "DB_MOTOR".COP2.Ctrl_Mode, Enable := "DB_MOTOR".COP2.Enable, Lock := "DB_MOTOR".COP2.Lock, Manual_Lock := "DB_MOTOR".COP2.Manual_Lock, Motor_Status := "DB_MOTOR".COP2.Status, Runtime_60s := "DB_MOTOR".COP2.Runtime_60s, Runtime_h := "DB_MOTOR".COP2.Runtime_h, Runtime_m := "DB_MOTOR".COP2.Runtime_m, Runtime_s := "DB_MOTOR".COP2.Runtime_s, Clock_temporary := "Clock_COP2", DQ_cmd => "DQ_COP2.Cmd")
   END_RUNG
   // the same network as SCL:
   "fc_Motor.Normal"(DI_Run := "DI_COP2.Run",
                     DI_Fault := "DI_COP2.Fault",
                     DI_Remote := "DI_COP2.Remote",
                     Ctrl_Mode := "DB_MOTOR".COP2.Ctrl_Mode,
                     Enable := "DB_MOTOR".COP2.Enable,
                     Lock := "DB_MOTOR".COP2.Lock,
                     Manual_Lock := "DB_MOTOR".COP2.Manual_Lock,
                     Motor_Status := "DB_MOTOR".COP2.Status,
                     Runtime_60s := "DB_MOTOR".COP2.Runtime_60s,
                     Runtime_h := "DB_MOTOR".COP2.Runtime_h,
                     Runtime_m := "DB_MOTOR".COP2.Runtime_m,
                     Runtime_s := "DB_MOTOR".COP2.Runtime_s,
                     Clock_temporary := "Clock_COP2",
                     DQ_cmd => "DQ_COP2.Cmd");
END_REGION

REGION Network 6: OSP
   RUNG wire#powerrail
      "fc_Motor.Normal"(DI_Run := "DI_OSP.Run", DI_Fault := "DI_OSP.Fault", DI_Remote := "DI_OSP.Remote", Ctrl_Mode := "DB_MOTOR".OSP.Ctrl_Mode, Enable := "DB_MOTOR".OSP.Enable, Lock := "DB_MOTOR".OSP.Lock, Manual_Lock := "DB_MOTOR".OSP.Manual_Lock, Motor_Status := "DB_MOTOR".OSP.Status, Runtime_60s := "DB_MOTOR".OSP.Runtime_60s, Runtime_h := "DB_MOTOR".OSP.Runtime_h, Runtime_m := "DB_MOTOR".OSP.Runtime_m, Runtime_s := "DB_MOTOR".OSP.Runtime_s, Clock_temporary := "Clock_OSP", DQ_cmd => "DQ_OSP.Cmd")
   END_RUNG
   // the same network as SCL:
   "fc_Motor.Normal"(DI_Run := "DI_OSP.Run",
                     DI_Fault := "DI_OSP.Fault",
                     DI_Remote := "DI_OSP.Remote",
                     Ctrl_Mode := "DB_MOTOR".OSP.Ctrl_Mode,
                     Enable := "DB_MOTOR".OSP.Enable,
                     Lock := "DB_MOTOR".OSP.Lock,
                     Manual_Lock := "DB_MOTOR".OSP.Manual_Lock,
                     Motor_Status := "DB_MOTOR".OSP.Status,
                     Runtime_60s := "DB_MOTOR".OSP.Runtime_60s,
                     Runtime_h := "DB_MOTOR".OSP.Runtime_h,
                     Runtime_m := "DB_MOTOR".OSP.Runtime_m,
                     Runtime_s := "DB_MOTOR".OSP.Runtime_s,
                     Clock_temporary := "Clock_OSP",
                     DQ_cmd => "DQ_OSP.Cmd");
END_REGION

REGION Network 7: ABC
   RUNG wire#powerrail
      "fc_Motor.Normal"(DI_Run := "DI_ABC.Run", DI_Fault := "DI_ABC.Fault", DI_Remote := "DI_ABC.Remote", Ctrl_Mode := "DB_MOTOR".ABC.Ctrl_Mode, Enable := "DB_MOTOR".ABC.Enable, Lock := "DB_MOTOR".ABC.Lock, Manual_Lock := "DB_MOTOR".ABC.Manual_Lock, Motor_Status := "DB_MOTOR".ABC.Status, Runtime_60s := "DB_MOTOR".ABC.Runtime_60s, Runtime_h := "DB_MOTOR".ABC.Runtime_h, Runtime_m := "DB_MOTOR".ABC.Runtime_m, Runtime_s := "DB_MOTOR".ABC.Runtime_s, Clock_temporary := "Clock_ABC", DQ_cmd => "DQ_ABC.Cmd")
   END_RUNG
   // the same network as SCL:
   "fc_Motor.Normal"(DI_Run := "DI_ABC.Run",
                     DI_Fault := "DI_ABC.Fault",
                     DI_Remote := "DI_ABC.Remote",
                     Ctrl_Mode := "DB_MOTOR".ABC.Ctrl_Mode,
                     Enable := "DB_MOTOR".ABC.Enable,
                     Lock := "DB_MOTOR".ABC.Lock,
                     Manual_Lock := "DB_MOTOR".ABC.Manual_Lock,
                     Motor_Status := "DB_MOTOR".ABC.Status,
                     Runtime_60s := "DB_MOTOR".ABC.Runtime_60s,
                     Runtime_h := "DB_MOTOR".ABC.Runtime_h,
                     Runtime_m := "DB_MOTOR".ABC.Runtime_m,
                     Runtime_s := "DB_MOTOR".ABC.Runtime_s,
                     Clock_temporary := "Clock_ABC",
                     DQ_cmd => "DQ_ABC.Cmd");
END_REGION

REGION Network 8: Reset runtime60s
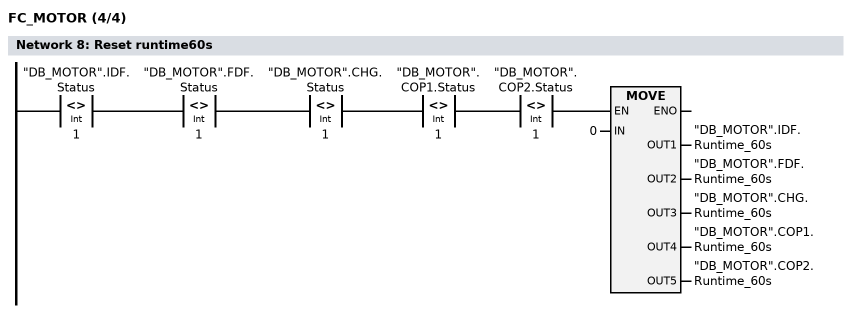
   RUNG wire#powerrail
      { S7_Templates := "SrcType := Int" } NE_Contact(in1 := "DB_MOTOR".IDF.Status, in2 := 1)
      { S7_Templates := "SrcType := Int" } NE_Contact(in1 := "DB_MOTOR".FDF.Status, in2 := 1)
      { S7_Templates := "SrcType := Int" } NE_Contact(in1 := "DB_MOTOR".CHG.Status, in2 := 1)
      { S7_Templates := "SrcType := Int" } NE_Contact(in1 := "DB_MOTOR".COP1.Status, in2 := 1)
      { S7_Templates := "SrcType := Int" } NE_Contact(in1 := "DB_MOTOR".COP2.Status, in2 := 1)
      Move(in := 0, out1 => "DB_MOTOR".IDF.Runtime_60s, out2 => "DB_MOTOR".FDF.Runtime_60s, out3 => "DB_MOTOR".CHG.Runtime_60s, out4 => "DB_MOTOR".COP1.Runtime_60s, out5 => "DB_MOTOR".COP2.Runtime_60s)
   END_RUNG
   // the same network as SCL:
   IF ("DB_MOTOR".IDF.Status <> 1) AND ("DB_MOTOR".FDF.Status <> 1) AND ("DB_MOTOR".CHG.Status <> 1) AND ("DB_MOTOR".COP1.Status <> 1) AND ("DB_MOTOR".COP2.Status <> 1) THEN
       "DB_MOTOR".IDF.Runtime_60s := 0;
       "DB_MOTOR".FDF.Runtime_60s := 0;
       "DB_MOTOR".CHG.Runtime_60s := 0;
       "DB_MOTOR".COP1.Runtime_60s := 0;
       "DB_MOTOR".COP2.Runtime_60s := 0;
   END_IF;
END_REGION
END_FUNCTION

FUNCTION "FC_INTERLOCK" : Void   // FC5, LAD
{ S7_Optimized_Access := 'TRUE' }
VERSION : 0.1
BEGIN

REGION Network 1: Tinh chenh ap dau
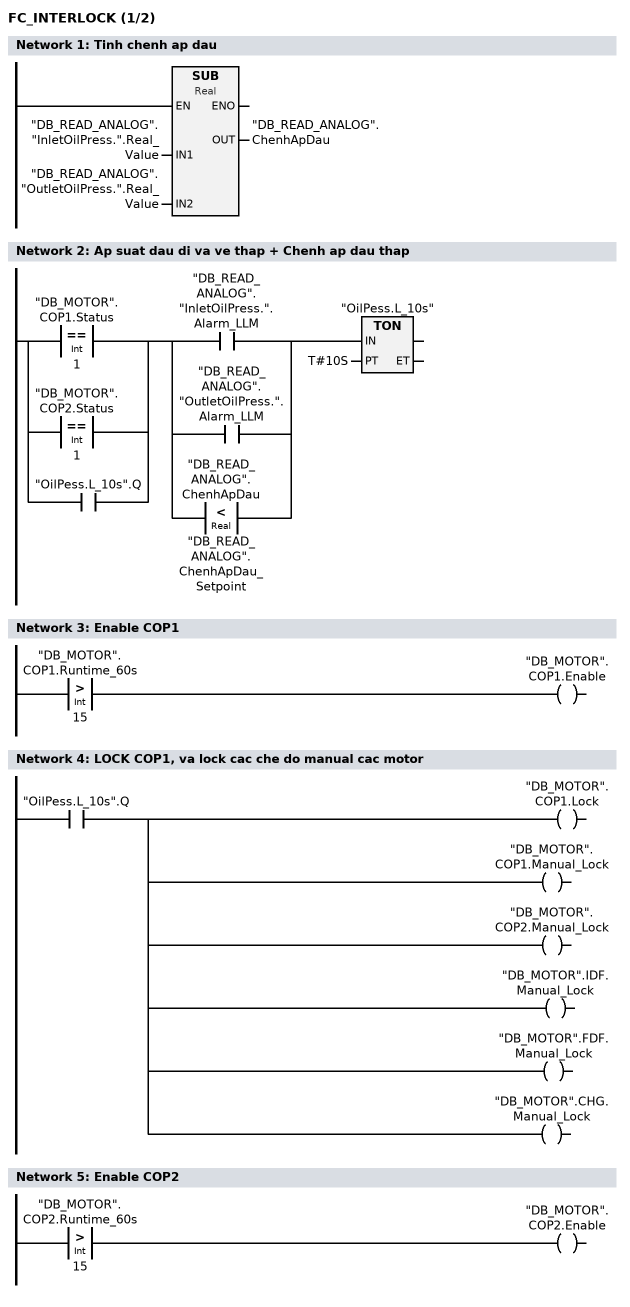
   RUNG wire#powerrail
      { S7_Templates := "SrcType := Real" } Sub(in1 := "DB_READ_ANALOG"."InletOilPress.".Real_Value, in2 := "DB_READ_ANALOG"."OutletOilPress.".Real_Value, out => "DB_READ_ANALOG".ChenhApDau)
   END_RUNG
   // the same network as SCL:
   "DB_READ_ANALOG".ChenhApDau := "DB_READ_ANALOG"."InletOilPress.".Real_Value - "DB_READ_ANALOG"."OutletOilPress.".Real_Value;
END_REGION

REGION Network 2: Ap suat dau di va ve thap + Chenh ap dau thap
   "OilPess.L_10s".TON(IN := (("DB_MOTOR".COP1.Status = 1) OR ("DB_MOTOR".COP2.Status = 1) OR "OilPess.L_10s".Q) AND ("DB_READ_ANALOG"."InletOilPress.".Alarm_LLM OR "DB_READ_ANALOG"."OutletOilPress.".Alarm_LLM OR ("DB_READ_ANALOG".ChenhApDau < "DB_READ_ANALOG".ChenhApDau_Setpoint)),
                       PT := T#10S);
END_REGION

REGION Network 3: Enable COP1
   RUNG wire#powerrail
      { S7_Templates := "SrcType := Int" } GT_Contact(in1 := "DB_MOTOR".COP1.Runtime_60s, in2 := 15)
      Coil( "DB_MOTOR".COP1.Enable )
   END_RUNG
   // the same network as SCL:
   "DB_MOTOR".COP1.Enable := "DB_MOTOR".COP1.Runtime_60s > 15;
END_REGION

REGION Network 4: LOCK COP1, va lock cac che do manual cac motor
   RUNG wire#powerrail
      Contact( "OilPess.L_10s".Q )
      wire#w1
      Coil( "DB_MOTOR".COP1.Lock )
   END_RUNG
   RUNG wire#w1
      Coil( "DB_MOTOR".COP1.Manual_Lock )
   END_RUNG
   RUNG wire#w1
      Coil( "DB_MOTOR".COP2.Manual_Lock )
   END_RUNG
   RUNG wire#w1
      Coil( "DB_MOTOR".IDF.Manual_Lock )
   END_RUNG
   RUNG wire#w1
      Coil( "DB_MOTOR".FDF.Manual_Lock )
   END_RUNG
   RUNG wire#w1
      Coil( "DB_MOTOR".CHG.Manual_Lock )
   END_RUNG
   // the same network as SCL:
   "DB_MOTOR".COP1.Lock := "OilPess.L_10s".Q;
   "DB_MOTOR".COP1.Manual_Lock := "OilPess.L_10s".Q;
   "DB_MOTOR".COP2.Manual_Lock := "OilPess.L_10s".Q;
   "DB_MOTOR".IDF.Manual_Lock := "OilPess.L_10s".Q;
   "DB_MOTOR".FDF.Manual_Lock := "OilPess.L_10s".Q;
   "DB_MOTOR".CHG.Manual_Lock := "OilPess.L_10s".Q;
END_REGION

REGION Network 5: Enable COP2
   RUNG wire#powerrail
      { S7_Templates := "SrcType := Int" } GT_Contact(in1 := "DB_MOTOR".COP2.Runtime_60s, in2 := 15)
      Coil( "DB_MOTOR".COP2.Enable )
   END_RUNG
   // the same network as SCL:
   "DB_MOTOR".COP2.Enable := "DB_MOTOR".COP2.Runtime_60s > 15;
END_REGION

REGION Network 6: LOCK COP2
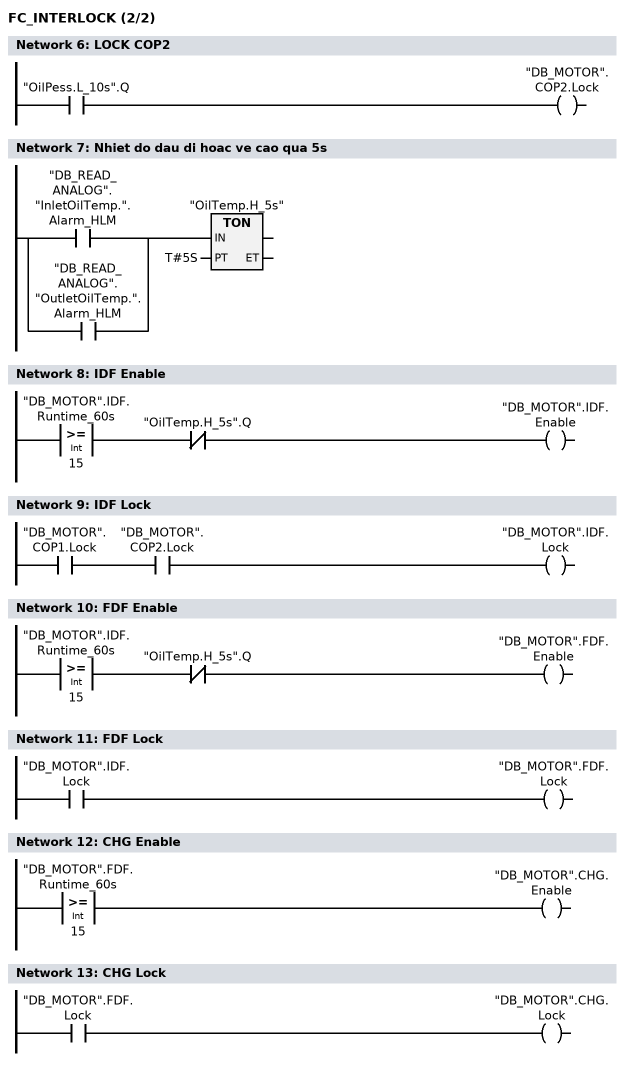
   RUNG wire#powerrail
      Contact( "OilPess.L_10s".Q )
      Coil( "DB_MOTOR".COP2.Lock )
   END_RUNG
   // the same network as SCL:
   "DB_MOTOR".COP2.Lock := "OilPess.L_10s".Q;
END_REGION

REGION Network 7: Nhiet do dau di hoac ve cao qua 5s
   "OilTemp.H_5s".TON(IN := "DB_READ_ANALOG"."InletOilTemp.".Alarm_HLM OR "DB_READ_ANALOG"."OutletOilTemp.".Alarm_HLM,
                      PT := T#5S);
END_REGION

REGION Network 8: IDF Enable
   RUNG wire#powerrail
      { S7_Templates := "SrcType := Int" } GE_Contact(in1 := "DB_MOTOR".IDF.Runtime_60s, in2 := 15)
      I_Contact( "OilTemp.H_5s".Q )
      Coil( "DB_MOTOR".IDF.Enable )
   END_RUNG
   // the same network as SCL:
   "DB_MOTOR".IDF.Enable := ("DB_MOTOR".IDF.Runtime_60s >= 15) AND NOT "OilTemp.H_5s".Q;
END_REGION

REGION Network 9: IDF Lock
   RUNG wire#powerrail
      Contact( "DB_MOTOR".COP1.Lock )
      Contact( "DB_MOTOR".COP2.Lock )
      Coil( "DB_MOTOR".IDF.Lock )
   END_RUNG
   // the same network as SCL:
   "DB_MOTOR".IDF.Lock := "DB_MOTOR".COP1.Lock AND "DB_MOTOR".COP2.Lock;
END_REGION

REGION Network 10: FDF Enable
   RUNG wire#powerrail
      { S7_Templates := "SrcType := Int" } GE_Contact(in1 := "DB_MOTOR".IDF.Runtime_60s, in2 := 15)
      I_Contact( "OilTemp.H_5s".Q )
      Coil( "DB_MOTOR".FDF.Enable )
   END_RUNG
   // the same network as SCL:
   "DB_MOTOR".FDF.Enable := ("DB_MOTOR".IDF.Runtime_60s >= 15) AND NOT "OilTemp.H_5s".Q;
END_REGION

REGION Network 11: FDF Lock
   RUNG wire#powerrail
      Contact( "DB_MOTOR".IDF.Lock )
      Coil( "DB_MOTOR".FDF.Lock )
   END_RUNG
   // the same network as SCL:
   "DB_MOTOR".FDF.Lock := "DB_MOTOR".IDF.Lock;
END_REGION

REGION Network 12: CHG Enable
   RUNG wire#powerrail
      { S7_Templates := "SrcType := Int" } GE_Contact(in1 := "DB_MOTOR".FDF.Runtime_60s, in2 := 15)
      Coil( "DB_MOTOR".CHG.Enable )
   END_RUNG
   // the same network as SCL:
   "DB_MOTOR".CHG.Enable := "DB_MOTOR".FDF.Runtime_60s >= 15;
END_REGION

REGION Network 13: CHG Lock
   RUNG wire#powerrail
      Contact( "DB_MOTOR".FDF.Lock )
      Coil( "DB_MOTOR".CHG.Lock )
   END_RUNG
   // the same network as SCL:
   "DB_MOTOR".CHG.Lock := "DB_MOTOR".FDF.Lock;
END_REGION
END_FUNCTION

FUNCTION "FC_WRITE_ANALOG" : Void   // FC8, LAD
{ S7_Optimized_Access := 'TRUE' }
VERSION : 0.1
BEGIN

REGION Network 1: xuat output hieu dieu khien IDF
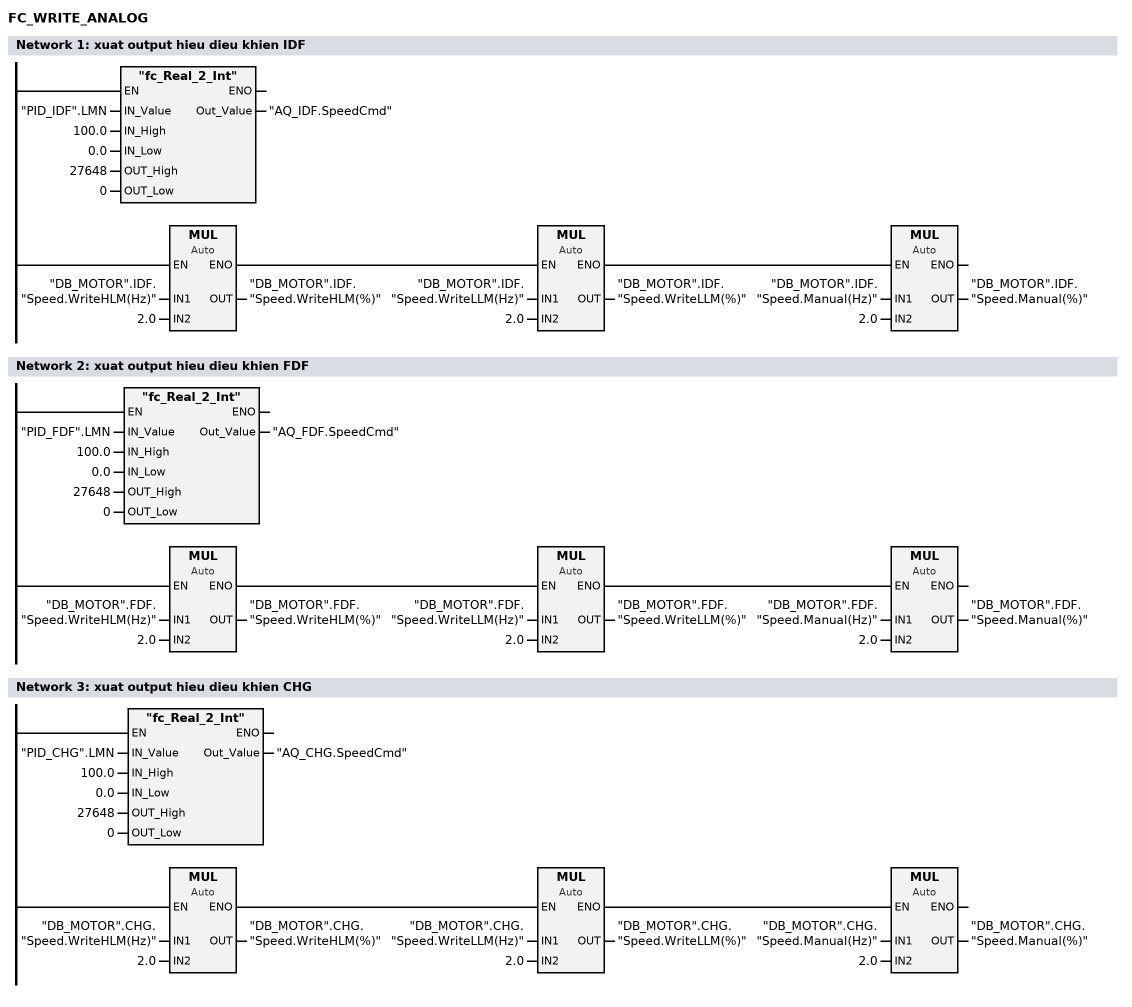
   RUNG wire#powerrail
      "fc_Real_2_Int"(IN_Value := "PID_IDF".LMN, IN_High := 100.0, IN_Low := 0.0, OUT_High := 27648, OUT_Low := 0, Out_Value => "AQ_IDF.SpeedCmd")
   END_RUNG
   RUNG wire#powerrail
      Mul(in1 := "DB_MOTOR".IDF."Speed.WriteHLM(Hz)", in2 := 2.0, out => "DB_MOTOR".IDF."Speed.WriteHLM(%)")
      Mul(in1 := "DB_MOTOR".IDF."Speed.WriteLLM(Hz)", in2 := 2.0, out => "DB_MOTOR".IDF."Speed.WriteLLM(%)")
      Mul(in1 := "DB_MOTOR".IDF."Speed.Manual(Hz)", in2 := 2.0, out => "DB_MOTOR".IDF."Speed.Manual(%)")
   END_RUNG
   // the same network as SCL:
   "fc_Real_2_Int"(IN_Value := "PID_IDF".LMN,
                   IN_High := 100.0,
                   IN_Low := 0.0,
                   OUT_High := 27648,
                   OUT_Low := 0,
                   Out_Value => "AQ_IDF.SpeedCmd");
   "DB_MOTOR".IDF."Speed.WriteHLM(%)" := "DB_MOTOR".IDF."Speed.WriteHLM(Hz)" * 2.0;
   "DB_MOTOR".IDF."Speed.WriteLLM(%)" := "DB_MOTOR".IDF."Speed.WriteLLM(Hz)" * 2.0;
   "DB_MOTOR".IDF."Speed.Manual(%)" := "DB_MOTOR".IDF."Speed.Manual(Hz)" * 2.0;
END_REGION

REGION Network 2: xuat output hieu dieu khien FDF
   RUNG wire#powerrail
      "fc_Real_2_Int"(IN_Value := "PID_FDF".LMN, IN_High := 100.0, IN_Low := 0.0, OUT_High := 27648, OUT_Low := 0, Out_Value => "AQ_FDF.SpeedCmd")
   END_RUNG
   RUNG wire#powerrail
      Mul(in1 := "DB_MOTOR".FDF."Speed.WriteHLM(Hz)", in2 := 2.0, out => "DB_MOTOR".FDF."Speed.WriteHLM(%)")
      Mul(in1 := "DB_MOTOR".FDF."Speed.WriteLLM(Hz)", in2 := 2.0, out => "DB_MOTOR".FDF."Speed.WriteLLM(%)")
      Mul(in1 := "DB_MOTOR".FDF."Speed.Manual(Hz)", in2 := 2.0, out => "DB_MOTOR".FDF."Speed.Manual(%)")
   END_RUNG
   // the same network as SCL:
   "fc_Real_2_Int"(IN_Value := "PID_FDF".LMN,
                   IN_High := 100.0,
                   IN_Low := 0.0,
                   OUT_High := 27648,
                   OUT_Low := 0,
                   Out_Value => "AQ_FDF.SpeedCmd");
   "DB_MOTOR".FDF."Speed.WriteHLM(%)" := "DB_MOTOR".FDF."Speed.WriteHLM(Hz)" * 2.0;
   "DB_MOTOR".FDF."Speed.WriteLLM(%)" := "DB_MOTOR".FDF."Speed.WriteLLM(Hz)" * 2.0;
   "DB_MOTOR".FDF."Speed.Manual(%)" := "DB_MOTOR".FDF."Speed.Manual(Hz)" * 2.0;
END_REGION

REGION Network 3: xuat output hieu dieu khien CHG
   RUNG wire#powerrail
      "fc_Real_2_Int"(IN_Value := "PID_CHG".LMN, IN_High := 100.0, IN_Low := 0.0, OUT_High := 27648, OUT_Low := 0, Out_Value => "AQ_CHG.SpeedCmd")
   END_RUNG
   RUNG wire#powerrail
      Mul(in1 := "DB_MOTOR".CHG."Speed.WriteHLM(Hz)", in2 := 2.0, out => "DB_MOTOR".CHG."Speed.WriteHLM(%)")
      Mul(in1 := "DB_MOTOR".CHG."Speed.WriteLLM(Hz)", in2 := 2.0, out => "DB_MOTOR".CHG."Speed.WriteLLM(%)")
      Mul(in1 := "DB_MOTOR".CHG."Speed.Manual(Hz)", in2 := 2.0, out => "DB_MOTOR".CHG."Speed.Manual(%)")
   END_RUNG
   // the same network as SCL:
   "fc_Real_2_Int"(IN_Value := "PID_CHG".LMN,
                   IN_High := 100.0,
                   IN_Low := 0.0,
                   OUT_High := 27648,
                   OUT_Low := 0,
                   Out_Value => "AQ_CHG.SpeedCmd");
   "DB_MOTOR".CHG."Speed.WriteHLM(%)" := "DB_MOTOR".CHG."Speed.WriteHLM(Hz)" * 2.0;
   "DB_MOTOR".CHG."Speed.WriteLLM(%)" := "DB_MOTOR".CHG."Speed.WriteLLM(Hz)" * 2.0;
   "DB_MOTOR".CHG."Speed.Manual(%)" := "DB_MOTOR".CHG."Speed.Manual(Hz)" * 2.0;
END_REGION
END_FUNCTION

ORGANIZATION_BLOCK "Main"   // OB1, LAD, ProgramCycle
TITLE = "Main Program Sweep (Cycle)"
{ S7_Optimized_Access := 'TRUE' }
VERSION : 0.1
BEGIN
END_ORGANIZATION_BLOCK

// folder: Function

FUNCTION "fc_Scale_Sensor" : Void   // FC1, SCL
{ S7_Optimized_Access := 'TRUE' }
VERSION : 0.1
   VAR_INPUT
      Input : Int;
      In_Low : Int;
      In_High : Int;
      Value_Low : Real;
      Value_High : Real;
      Ratio : Real;
      Bias : Real;
   END_VAR
   VAR_OUTPUT
      Value : Real;
      Error_Input : Bool;
   END_VAR
BEGIN
   IF (#In_Low < #In_High) AND (#Value_Low < #Value_High) THEN
       #Value := (INT_TO_REAL(#Input - #In_Low) / INT_TO_REAL(#In_High - #In_Low) * (#Value_High - #Value_Low) + #Value_Low) * #Ratio + #Bias;
       #Error_Input := FALSE;
   ELSE
       #Value := 0;
       #Error_Input := TRUE;
   END_IF;
END_FUNCTION

FUNCTION "fc_Read_Speed" : Void   // FC7, SCL
{ S7_Optimized_Access := 'TRUE' }
VERSION : 0.1
   VAR_INPUT
      Input : Int;
      In_Low : Int;
      In_High : Int;
      Value_Low : Real;
      Value_High : Real;
      Ratio : Real;
      Bias : Real;
   END_VAR
   VAR_OUTPUT
      Value : Real;
   END_VAR
BEGIN
   IF (#In_Low < #In_High) AND (#Value_Low < #Value_High) THEN
       #Value := (INT_TO_REAL(#Input - #In_Low) / INT_TO_REAL(#In_High - #In_Low) * (#Value_High - #Value_Low) + #Value_Low) * #Ratio + #Bias;

   ELSE
       #Value := 0;

   END_IF;
END_FUNCTION

FUNCTION "fc_AnalogOutput" : Void   // FC9, LAD
{ S7_Optimized_Access := 'TRUE' }
VERSION : 0.1
   VAR_INPUT
      Man_On : Bool;
      Man_Value : Real;
      PID_Value : Real;
      HLM_Value : Real;
      LLM_Value : Real;
   END_VAR
   VAR_OUTPUT
      Analoge_Out : Int;
      SCADA_Value : Real;
   END_VAR
   VAR_TEMP
      Temp_Real : Real;
   END_VAR
   VAR_TEMP   // added for the SCL form of the ladder/FBD networks
      _w1 : Bool;
      _w2 : Bool;
   END_VAR
BEGIN

REGION Network 1
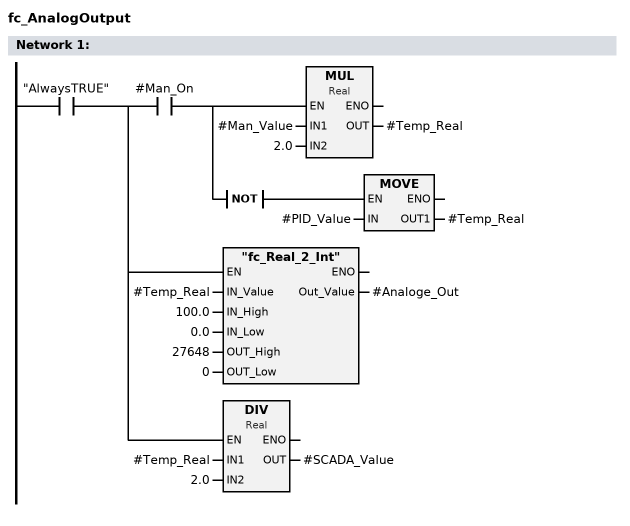
   RUNG wire#powerrail
      Contact( "AlwaysTRUE" )
      wire#w1
      Contact( #Man_On )
      wire#w2
      { S7_Templates := "SrcType := Real"; S7_GenerateENO := "TRUE" } Mul(in1 := #Man_Value, in2 := 2.0, out => #Temp_Real)
   END_RUNG
   RUNG wire#w2
      Not()
      Move(in := #PID_Value, out1 => #Temp_Real)
   END_RUNG
   RUNG wire#w1
      "fc_Real_2_Int"(IN_Value := #Temp_Real, IN_High := 100.0, IN_Low := 0.0, OUT_High := 27648, OUT_Low := 0, Out_Value => #Analoge_Out)
   END_RUNG
   RUNG wire#w1
      { S7_Templates := "SrcType := Real"; S7_GenerateENO := "TRUE" } Div(in1 := #Temp_Real, in2 := 2.0, out => #SCADA_Value)
   END_RUNG
   // the same network as SCL:
   #_w1 := "AlwaysTRUE" AND #Man_On;
   IF #_w1 THEN #Temp_Real := #Man_Value * 2.0; END_IF;
   IF NOT #_w1 THEN #Temp_Real := #PID_Value; END_IF;
   #_w2 := "AlwaysTRUE";
   IF #_w2 THEN
       "fc_Real_2_Int"(IN_Value := #Temp_Real,
                       IN_High := 100.0,
                       IN_Low := 0.0,
                       OUT_High := 27648,
                       OUT_Low := 0,
                       Out_Value => #Analoge_Out);
       #SCADA_Value := #Temp_Real / 2.0;
   END_IF;
END_REGION
END_FUNCTION

FUNCTION "fc_Real_2_Real" : Void   // FC10, SCL
{ S7_Optimized_Access := 'TRUE' }
VERSION : 0.1
   VAR_INPUT
      IN_Value : Real;
      IN_High : Real;
      IN_Low : Real;
      OUT_High : Real;
      OUT_Low : Real;
   END_VAR
   VAR_OUTPUT
      Out_Value : Real;
   END_VAR
BEGIN
   #Out_Value := ((#IN_Value - #IN_Low) / (#IN_High - #IN_Low)) * (#OUT_High - #OUT_Low) + #OUT_Low;
END_FUNCTION

FUNCTION "fc_Real_2_Int" : Void   // FC11, SCL
{ S7_Optimized_Access := 'TRUE' }
VERSION : 0.1
   VAR_INPUT
      IN_Value : Real;
      IN_High : Real;
      IN_Low : Real;
      OUT_High : Int;
      OUT_Low : Int;
   END_VAR
   VAR_OUTPUT
      Out_Value : Int;
   END_VAR
   VAR_TEMP
      Temp_Real : Real;
   END_VAR
BEGIN
   #Temp_Real := ((#IN_Value - #IN_Low) / (#IN_High - #IN_Low)) * INT_TO_REAL(#OUT_High - #OUT_Low);
   #Out_Value := REAL_TO_INT(#Temp_Real) + #OUT_Low;
END_FUNCTION

FUNCTION "fc_Motor.VFD" : Void   // FC12, LAD
{ S7_Optimized_Access := 'TRUE' }
VERSION : 0.1
   VAR_INPUT
      DI_Run : Bool;
      DI_Fault : Bool;
      DI_Remote : Bool;
      Ctrl_Mode : Int;
      Enable : Bool;
      Lock : Bool;
      Manual_Lock : Bool;
      P : Real;
      P_factor : Real;
      I : Real;
      D : Real;
   END_VAR
   VAR_OUTPUT
      DQ_cmd : Bool;
      PID_Gain : Real;
      PID_Ti : Time;
      PID_Td : Time;
   END_VAR
   VAR_IN_OUT
      Motor_Status : Int;
      Runtime_60s : Int;
      Runtime_h : Int;
      Runtime_m : Int;
      Runtime_s : Int;
      Clock_temporary : Bool;   // Mx.x
   END_VAR
   VAR_TEMP   // added for the SCL form of the ladder/FBD networks
      _w1 : Bool;
   END_VAR
BEGIN

REGION Network 1: Status
   // Status: -1.Fault; 0.Stop; 1.Run
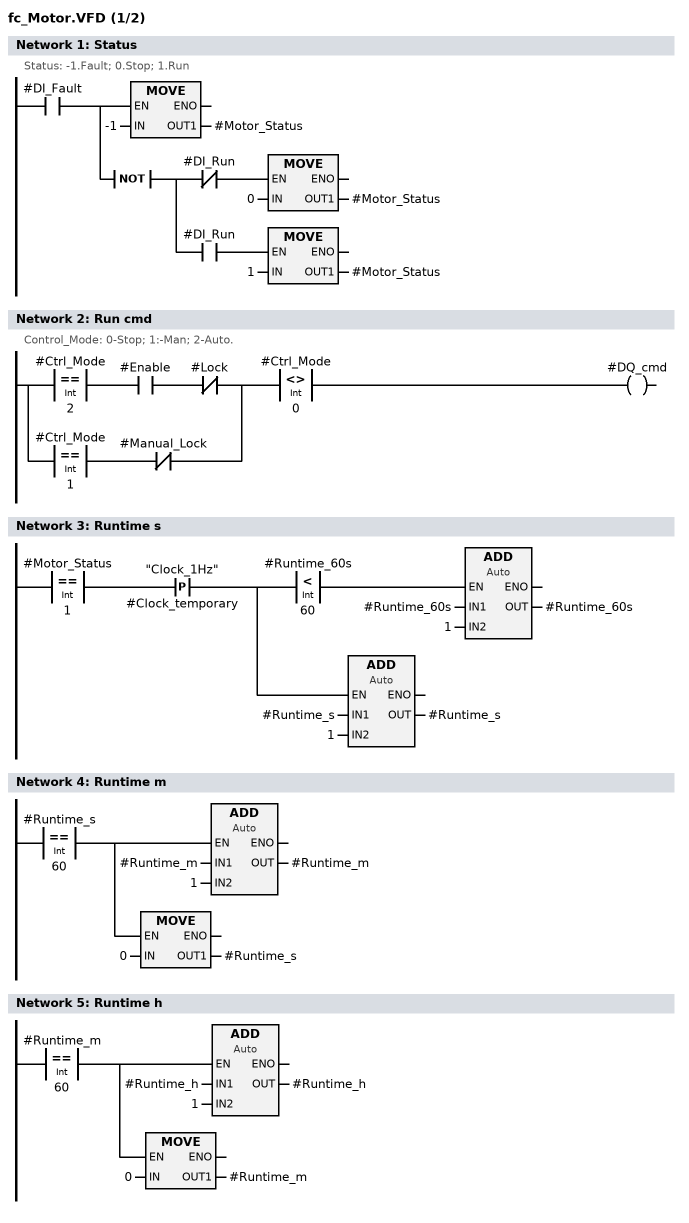
   RUNG wire#powerrail
      Contact( #DI_Fault )
      wire#w1
      Move(in := -1, out1 => #Motor_Status)
   END_RUNG
   RUNG wire#w1
      Not()
      wire#w2
      I_Contact( #DI_Run )
      Move(in := 0, out1 => #Motor_Status)
   END_RUNG
   RUNG wire#w2
      Contact( #DI_Run )
      Move(in := 1, out1 => #Motor_Status)
   END_RUNG
   // the same network as SCL:
   IF #DI_Fault THEN #Motor_Status := -1; END_IF;
   IF NOT #DI_Fault AND NOT #DI_Run THEN #Motor_Status := 0; END_IF;
   IF NOT #DI_Fault AND #DI_Run THEN #Motor_Status := 1; END_IF;
END_REGION

REGION Network 2: Run cmd
   // Control_Mode: 0-Stop; 1:-Man; 2-Auto.
   RUNG wire#powerrail
      { S7_Templates := "SrcType := Int" } EQ_Contact(in1 := #Ctrl_Mode, in2 := 2)
      Contact( #Enable )
      I_Contact( #Lock )
      wire#w1
      { S7_Templates := "SrcType := Int" } NE_Contact(in1 := #Ctrl_Mode, in2 := 0)
      Coil( #DQ_cmd )
   END_RUNG
   RUNG wire#powerrail
      { S7_Templates := "SrcType := Int" } EQ_Contact(in1 := #Ctrl_Mode, in2 := 1)
      I_Contact( #Manual_Lock )
   END_RUNG wire#w1
   // the same network as SCL:
   #DQ_cmd := (((#Ctrl_Mode = 2) AND #Enable AND NOT #Lock) OR ((#Ctrl_Mode = 1) AND NOT #Manual_Lock)) AND (#Ctrl_Mode <> 0);
END_REGION

REGION Network 3: Runtime s
   RUNG wire#powerrail
      { S7_Templates := "SrcType := Int" } EQ_Contact(in1 := #Motor_Status, in2 := 1)
      P_Contact(operand := "Clock_1Hz", bit := #Clock_temporary)
      wire#w1
      { S7_Templates := "SrcType := Int" } LT_Contact(in1 := #Runtime_60s, in2 := 60)
      Add(in1 := #Runtime_60s, in2 := 1, out => #Runtime_60s)
   END_RUNG
   RUNG wire#w1
      Add(in1 := #Runtime_s, in2 := 1, out => #Runtime_s)
   END_RUNG
   // the same network as SCL:
   #_w1 := (#Motor_Status = 1) AND "Clock_1Hz" AND NOT #Clock_temporary;   // rising edge of "Clock_1Hz"
   #Clock_temporary := "Clock_1Hz";
   IF #_w1 AND (#Runtime_60s < 60) THEN #Runtime_60s := #Runtime_60s + 1; END_IF;
   IF #_w1 THEN #Runtime_s := #Runtime_s + 1; END_IF;
END_REGION

REGION Network 4: Runtime m
   RUNG wire#powerrail
      { S7_Templates := "SrcType := Int" } EQ_Contact(in1 := #Runtime_s, in2 := 60)
      wire#w1
      Add(in1 := #Runtime_m, in2 := 1, out => #Runtime_m)
   END_RUNG
   RUNG wire#w1
      Move(in := 0, out1 => #Runtime_s)
   END_RUNG
   // the same network as SCL:
   IF #Runtime_s = 60 THEN
       #Runtime_m := #Runtime_m + 1;
       #Runtime_s := 0;
   END_IF;
END_REGION

REGION Network 5: Runtime h
   RUNG wire#powerrail
      { S7_Templates := "SrcType := Int" } EQ_Contact(in1 := #Runtime_m, in2 := 60)
      wire#w1
      Add(in1 := #Runtime_h, in2 := 1, out => #Runtime_h)
   END_RUNG
   RUNG wire#w1
      Move(in := 0, out1 => #Runtime_m)
   END_RUNG
   // the same network as SCL:
   IF #Runtime_m = 60 THEN
       #Runtime_h := #Runtime_h + 1;
       #Runtime_m := 0;
   END_IF;
END_REGION

REGION Network 6: Xu li tran bo nho
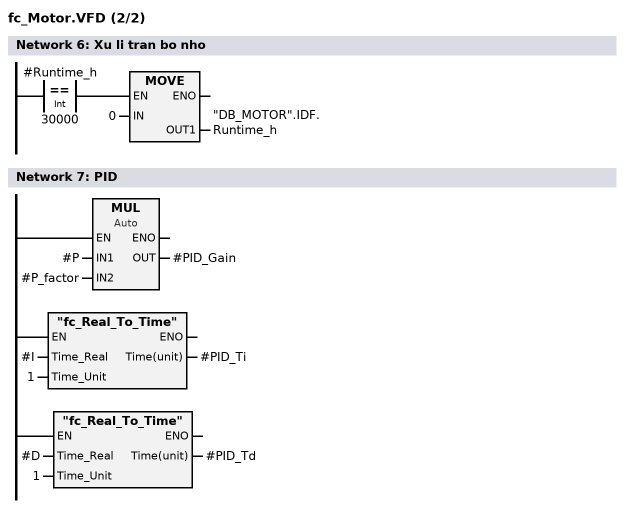
   RUNG wire#powerrail
      { S7_Templates := "SrcType := Int" } EQ_Contact(in1 := #Runtime_h, in2 := 30000)
      Move(in := 0, out1 => "DB_MOTOR".IDF.Runtime_h)
   END_RUNG
   // the same network as SCL:
   IF #Runtime_h = 30000 THEN "DB_MOTOR".IDF.Runtime_h := 0; END_IF;
END_REGION

REGION Network 7: PID
   RUNG wire#powerrail
      Mul(in1 := #P, in2 := #P_factor, out => #PID_Gain)
   END_RUNG
   RUNG wire#powerrail
      "fc_Real_To_Time"(Time_Real := #I, Time_Unit := 1, "Time(unit)" => #PID_Ti)
   END_RUNG
   RUNG wire#powerrail
      "fc_Real_To_Time"(Time_Real := #D, Time_Unit := 1, "Time(unit)" => #PID_Td)
   END_RUNG
   // the same network as SCL:
   #PID_Gain := #P * #P_factor;
   "fc_Real_To_Time"(Time_Real := #I, Time_Unit := 1, "Time(unit)" => #PID_Ti);
   "fc_Real_To_Time"(Time_Real := #D, Time_Unit := 1, "Time(unit)" => #PID_Td);
END_REGION
END_FUNCTION

FUNCTION "fc_Real_To_Time" : Void   // FC13, SCL
{ S7_Optimized_Access := 'FALSE' }
VERSION : 0.1
   VAR_INPUT
      Time_Real : Real;
      Time_Unit : Int;   // ms_s(default)_m_h
   END_VAR
   VAR_OUTPUT
      "Time(unit)" : Time;
   END_VAR
   VAR_TEMP
      "DW(unit)" : DInt;
   END_VAR
BEGIN
   CASE #Time_Unit OF
       0:  //ms
           #"DW(unit)" := REAL_TO_DINT(#Time_Real);
           ;
       1: //s
           #"DW(unit)" := REAL_TO_DINT(#Time_Real * 1000);
           ;
       2:  //m
           #"DW(unit)" := REAL_TO_DINT(#Time_Real * 60000);
           ;
       3:  //h
           #"DW(unit)" := REAL_TO_DINT(#Time_Real * 3600000);
           ;
       ELSE
           #"DW(unit)" := REAL_TO_DINT(#Time_Real * 1000);
   END_CASE;

   #"Time(unit)" := DINT_TO_TIME(#"DW(unit)");
END_FUNCTION

FUNCTION "fc_Motor.2Directions" : Void   // FC14, LAD
{ S7_Optimized_Access := 'TRUE' }
VERSION : 0.1
   VAR_INPUT
      DI_RunForward : Bool;
      DI_RunReverse : Bool;
      DI_Fault : Bool;
      DI_Remote : Bool;
      Ctrl_Mode : Int;
      Enable : Bool;
      Lock : Bool;
      Manual_Lock : Bool;
      "Forward/Reverse" : Bool;   // 1: Forward; 0: Reverse.
   END_VAR
   VAR_OUTPUT
      "DQ_Forward.cmd" : Bool;
      "DQ_Reverse.cmd" : Bool;
   END_VAR
   VAR_IN_OUT
      Motor_Status : Int;
      Runtime_60s : Int;
      Runtime_h : Int;
      Runtime_m : Int;
      Runtime_s : Int;
      Clock_temporary : Bool;
   END_VAR
   VAR_TEMP   // added for the SCL form of the ladder/FBD networks
      _w1 : Bool;
   END_VAR
BEGIN

REGION Network 1: Status
   // Status: -1.Fault; 0.Stop; 1.Run
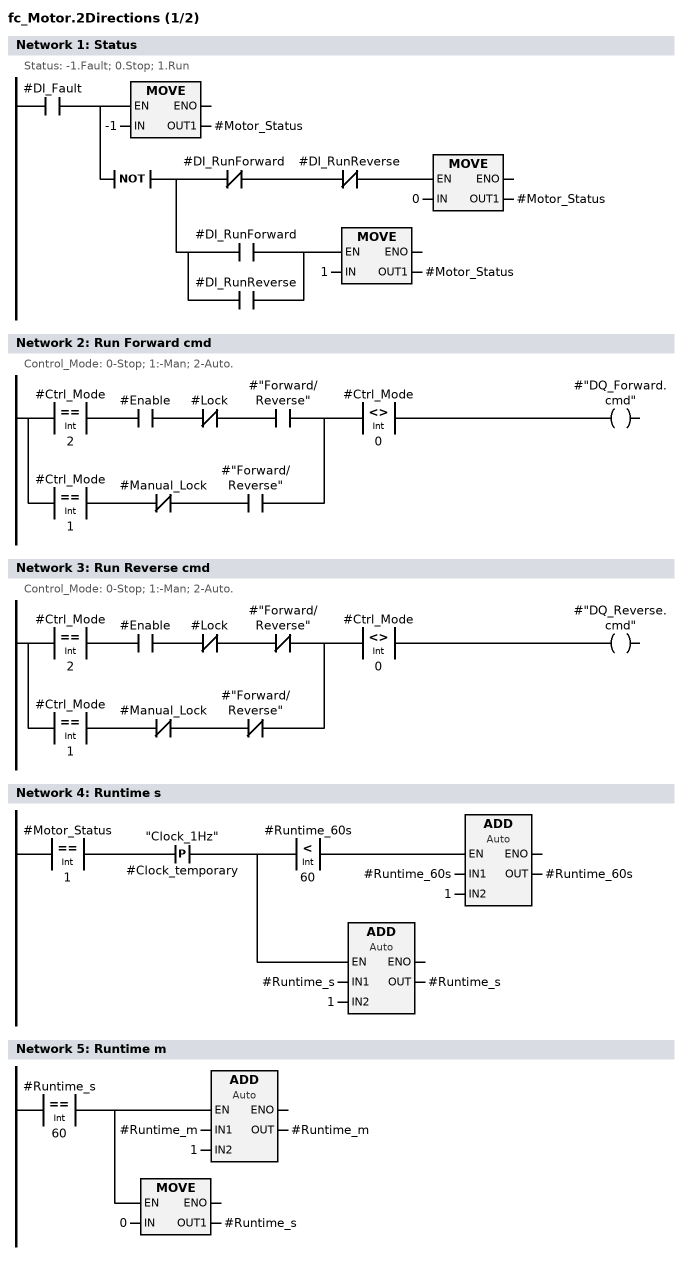
   RUNG wire#powerrail
      Contact( #DI_Fault )
      wire#w1
      Move(in := -1, out1 => #Motor_Status)
   END_RUNG
   RUNG wire#w1
      Not()
      wire#w2
      I_Contact( #DI_RunForward )
      I_Contact( #DI_RunReverse )
      Move(in := 0, out1 => #Motor_Status)
   END_RUNG
   RUNG wire#w2
      Contact( #DI_RunForward )
      wire#w3
      Move(in := 1, out1 => #Motor_Status)
   END_RUNG
   RUNG wire#w2
      Contact( #DI_RunReverse )
   END_RUNG wire#w3
   // the same network as SCL:
   IF #DI_Fault THEN #Motor_Status := -1; END_IF;
   IF NOT #DI_Fault AND NOT #DI_RunForward AND NOT #DI_RunReverse THEN #Motor_Status := 0; END_IF;
   IF NOT #DI_Fault AND (#DI_RunForward OR #DI_RunReverse) THEN #Motor_Status := 1; END_IF;
END_REGION

REGION Network 2: Run Forward cmd
   // Control_Mode: 0-Stop; 1:-Man; 2-Auto.
   RUNG wire#powerrail
      { S7_Templates := "SrcType := Int" } EQ_Contact(in1 := #Ctrl_Mode, in2 := 2)
      Contact( #Enable )
      I_Contact( #Lock )
      Contact( #"Forward/Reverse" )
      wire#w1
      { S7_Templates := "SrcType := Int" } NE_Contact(in1 := #Ctrl_Mode, in2 := 0)
      Coil( #"DQ_Forward.cmd" )
   END_RUNG
   RUNG wire#powerrail
      { S7_Templates := "SrcType := Int" } EQ_Contact(in1 := #Ctrl_Mode, in2 := 1)
      I_Contact( #Manual_Lock )
      Contact( #"Forward/Reverse" )
   END_RUNG wire#w1
   // the same network as SCL:
   #"DQ_Forward.cmd" := (((#Ctrl_Mode = 2) AND #Enable AND NOT #Lock AND #"Forward/Reverse") OR ((#Ctrl_Mode = 1) AND NOT #Manual_Lock AND #"Forward/Reverse")) AND (#Ctrl_Mode <> 0);
END_REGION

REGION Network 3: Run Reverse cmd
   // Control_Mode: 0-Stop; 1:-Man; 2-Auto.
   RUNG wire#powerrail
      { S7_Templates := "SrcType := Int" } EQ_Contact(in1 := #Ctrl_Mode, in2 := 2)
      Contact( #Enable )
      I_Contact( #Lock )
      I_Contact( #"Forward/Reverse" )
      wire#w1
      { S7_Templates := "SrcType := Int" } NE_Contact(in1 := #Ctrl_Mode, in2 := 0)
      Coil( #"DQ_Reverse.cmd" )
   END_RUNG
   RUNG wire#powerrail
      { S7_Templates := "SrcType := Int" } EQ_Contact(in1 := #Ctrl_Mode, in2 := 1)
      I_Contact( #Manual_Lock )
      I_Contact( #"Forward/Reverse" )
   END_RUNG wire#w1
   // the same network as SCL:
   #"DQ_Reverse.cmd" := (((#Ctrl_Mode = 2) AND #Enable AND NOT #Lock AND NOT #"Forward/Reverse") OR ((#Ctrl_Mode = 1) AND NOT #Manual_Lock AND NOT #"Forward/Reverse")) AND (#Ctrl_Mode <> 0);
END_REGION

REGION Network 4: Runtime s
   RUNG wire#powerrail
      { S7_Templates := "SrcType := Int" } EQ_Contact(in1 := #Motor_Status, in2 := 1)
      P_Contact(operand := "Clock_1Hz", bit := #Clock_temporary)
      wire#w1
      { S7_Templates := "SrcType := Int" } LT_Contact(in1 := #Runtime_60s, in2 := 60)
      Add(in1 := #Runtime_60s, in2 := 1, out => #Runtime_60s)
   END_RUNG
   RUNG wire#w1
      Add(in1 := #Runtime_s, in2 := 1, out => #Runtime_s)
   END_RUNG
   // the same network as SCL:
   #_w1 := (#Motor_Status = 1) AND "Clock_1Hz" AND NOT #Clock_temporary;   // rising edge of "Clock_1Hz"
   #Clock_temporary := "Clock_1Hz";
   IF #_w1 AND (#Runtime_60s < 60) THEN #Runtime_60s := #Runtime_60s + 1; END_IF;
   IF #_w1 THEN #Runtime_s := #Runtime_s + 1; END_IF;
END_REGION

REGION Network 5: Runtime m
   RUNG wire#powerrail
      { S7_Templates := "SrcType := Int" } EQ_Contact(in1 := #Runtime_s, in2 := 60)
      wire#w1
      Add(in1 := #Runtime_m, in2 := 1, out => #Runtime_m)
   END_RUNG
   RUNG wire#w1
      Move(in := 0, out1 => #Runtime_s)
   END_RUNG
   // the same network as SCL:
   IF #Runtime_s = 60 THEN
       #Runtime_m := #Runtime_m + 1;
       #Runtime_s := 0;
   END_IF;
END_REGION

REGION Network 6: Runtime h
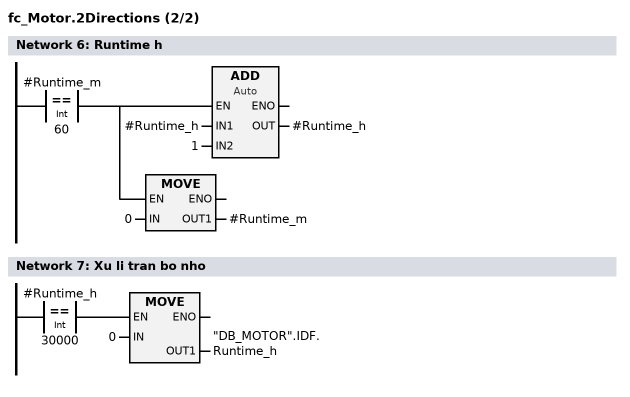
   RUNG wire#powerrail
      { S7_Templates := "SrcType := Int" } EQ_Contact(in1 := #Runtime_m, in2 := 60)
      wire#w1
      Add(in1 := #Runtime_h, in2 := 1, out => #Runtime_h)
   END_RUNG
   RUNG wire#w1
      Move(in := 0, out1 => #Runtime_m)
   END_RUNG
   // the same network as SCL:
   IF #Runtime_m = 60 THEN
       #Runtime_h := #Runtime_h + 1;
       #Runtime_m := 0;
   END_IF;
END_REGION

REGION Network 7: Xu li tran bo nho
   RUNG wire#powerrail
      { S7_Templates := "SrcType := Int" } EQ_Contact(in1 := #Runtime_h, in2 := 30000)
      Move(in := 0, out1 => "DB_MOTOR".IDF.Runtime_h)
   END_RUNG
   // the same network as SCL:
   IF #Runtime_h = 30000 THEN "DB_MOTOR".IDF.Runtime_h := 0; END_IF;
END_REGION
END_FUNCTION

FUNCTION "fc_Motor.Normal" : Void   // FC15, LAD
{ S7_Optimized_Access := 'TRUE' }
VERSION : 0.1
   VAR_INPUT
      DI_Run : Bool;
      DI_Fault : Bool;
      DI_Remote : Bool;
      Ctrl_Mode : Int;
      Enable : Bool;
      Lock : Bool;
      Manual_Lock : Bool;
   END_VAR
   VAR_OUTPUT
      DQ_cmd : Bool;
   END_VAR
   VAR_IN_OUT
      Motor_Status : Int;
      Runtime_60s : Int;
      Runtime_h : Int;
      Runtime_m : Int;
      Runtime_s : Int;
      Clock_temporary : Bool;
   END_VAR
   VAR_TEMP   // added for the SCL form of the ladder/FBD networks
      _w1 : Bool;
   END_VAR
BEGIN

REGION Network 1: Status
   // Status: -1.Fault; 0.Stop; 1.Run
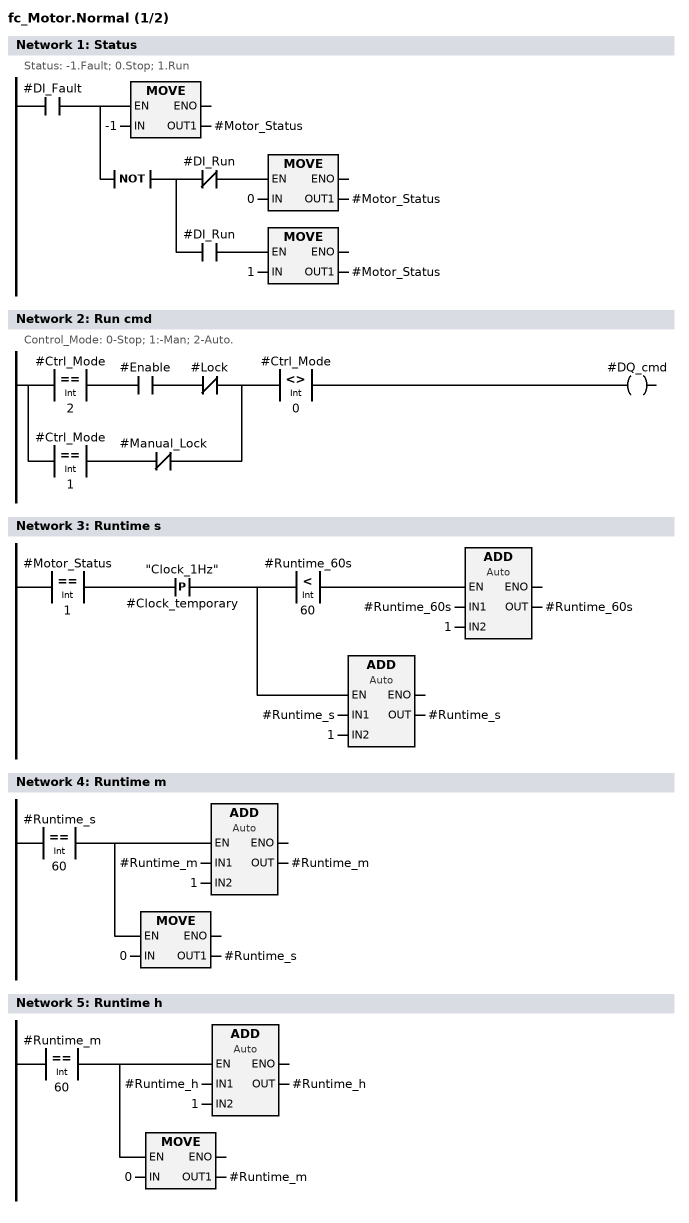
   RUNG wire#powerrail
      Contact( #DI_Fault )
      wire#w1
      Move(in := -1, out1 => #Motor_Status)
   END_RUNG
   RUNG wire#w1
      Not()
      wire#w2
      I_Contact( #DI_Run )
      Move(in := 0, out1 => #Motor_Status)
   END_RUNG
   RUNG wire#w2
      Contact( #DI_Run )
      Move(in := 1, out1 => #Motor_Status)
   END_RUNG
   // the same network as SCL:
   IF #DI_Fault THEN #Motor_Status := -1; END_IF;
   IF NOT #DI_Fault AND NOT #DI_Run THEN #Motor_Status := 0; END_IF;
   IF NOT #DI_Fault AND #DI_Run THEN #Motor_Status := 1; END_IF;
END_REGION

REGION Network 2: Run cmd
   // Control_Mode: 0-Stop; 1:-Man; 2-Auto.
   RUNG wire#powerrail
      { S7_Templates := "SrcType := Int" } EQ_Contact(in1 := #Ctrl_Mode, in2 := 2)
      Contact( #Enable )
      I_Contact( #Lock )
      wire#w1
      { S7_Templates := "SrcType := Int" } NE_Contact(in1 := #Ctrl_Mode, in2 := 0)
      Coil( #DQ_cmd )
   END_RUNG
   RUNG wire#powerrail
      { S7_Templates := "SrcType := Int" } EQ_Contact(in1 := #Ctrl_Mode, in2 := 1)
      I_Contact( #Manual_Lock )
   END_RUNG wire#w1
   // the same network as SCL:
   #DQ_cmd := (((#Ctrl_Mode = 2) AND #Enable AND NOT #Lock) OR ((#Ctrl_Mode = 1) AND NOT #Manual_Lock)) AND (#Ctrl_Mode <> 0);
END_REGION

REGION Network 3: Runtime s
   RUNG wire#powerrail
      { S7_Templates := "SrcType := Int" } EQ_Contact(in1 := #Motor_Status, in2 := 1)
      P_Contact(operand := "Clock_1Hz", bit := #Clock_temporary)
      wire#w1
      { S7_Templates := "SrcType := Int" } LT_Contact(in1 := #Runtime_60s, in2 := 60)
      Add(in1 := #Runtime_60s, in2 := 1, out => #Runtime_60s)
   END_RUNG
   RUNG wire#w1
      Add(in1 := #Runtime_s, in2 := 1, out => #Runtime_s)
   END_RUNG
   // the same network as SCL:
   #_w1 := (#Motor_Status = 1) AND "Clock_1Hz" AND NOT #Clock_temporary;   // rising edge of "Clock_1Hz"
   #Clock_temporary := "Clock_1Hz";
   IF #_w1 AND (#Runtime_60s < 60) THEN #Runtime_60s := #Runtime_60s + 1; END_IF;
   IF #_w1 THEN #Runtime_s := #Runtime_s + 1; END_IF;
END_REGION

REGION Network 4: Runtime m
   RUNG wire#powerrail
      { S7_Templates := "SrcType := Int" } EQ_Contact(in1 := #Runtime_s, in2 := 60)
      wire#w1
      Add(in1 := #Runtime_m, in2 := 1, out => #Runtime_m)
   END_RUNG
   RUNG wire#w1
      Move(in := 0, out1 => #Runtime_s)
   END_RUNG
   // the same network as SCL:
   IF #Runtime_s = 60 THEN
       #Runtime_m := #Runtime_m + 1;
       #Runtime_s := 0;
   END_IF;
END_REGION

REGION Network 5: Runtime h
   RUNG wire#powerrail
      { S7_Templates := "SrcType := Int" } EQ_Contact(in1 := #Runtime_m, in2 := 60)
      wire#w1
      Add(in1 := #Runtime_h, in2 := 1, out => #Runtime_h)
   END_RUNG
   RUNG wire#w1
      Move(in := 0, out1 => #Runtime_m)
   END_RUNG
   // the same network as SCL:
   IF #Runtime_m = 60 THEN
       #Runtime_h := #Runtime_h + 1;
       #Runtime_m := 0;
   END_IF;
END_REGION

REGION Network 6: Xu li tran bo nho
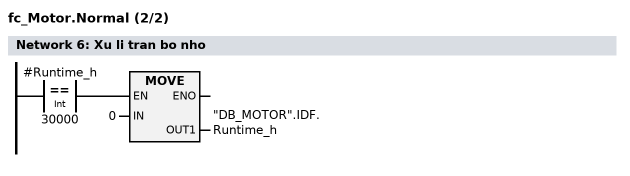
   RUNG wire#powerrail
      { S7_Templates := "SrcType := Int" } EQ_Contact(in1 := #Runtime_h, in2 := 30000)
      Move(in := 0, out1 => "DB_MOTOR".IDF.Runtime_h)
   END_RUNG
   // the same network as SCL:
   IF #Runtime_h = 30000 THEN "DB_MOTOR".IDF.Runtime_h := 0; END_IF;
END_REGION
END_FUNCTION